LIN {X 0,Y 469.68,Z 331.264,A -85,B 0,C 180,E1 -7635.818,E2 -7635.818} C_VEL
LIN {X 0,Y 469.232,Z 342.492,A -85,B 0,C 180,E1 -7636.5,E2 -7636.5} C_VEL
LIN {X 0,Y 468.814,Z 353.33,A -85,B 0,C 180,E1 -7637.334,E2 -7637.334} C_VEL
LIN {X 0,Y 468.372,Z 363.607,A -85,B 0,C 180,E1 -7638.314,E2 -7638.314} C_VEL
LIN {X 0,Y 467.885,Z 372.795,A -85,B 0,C 180,E1 -7639.398,E2 -7639.398} C_VEL
LIN {X 0,Y 467.445,Z 381.696,A -85,B 0,C 180,E1 -7640.7,E2 -7640.7} C_VEL
LIN {X 0,Y 467.091,Z 388.855,A -85,B 0,C 180,E1 -7642.001,E2 -7642.001} C_VEL
LIN {X 0,Y 466.869,Z 395.228,A -85,B 0,C 180,E1 -7643.48,E2 -7643.48} C_VEL
LIN {X 0,Y 466.783,Z 399.68,A -85,B 0,C 180,E1 -7644.818,E2 -7644.818} C_VEL
LIN {X 0,Y 466.662,Z 401.961,A -85,B 0,C 180,E1 -7645.683,E2 -7645.683} C_VEL
LIN {X 0,Y 466.695,Z 403.809,A -85,B 0,C 180,E1 -7646.548,E2 -7646.548} C_VEL
LIN {X 0,Y 466.646,Z 405.194,A -85,B 0,C 180,E1 -7647.412,E2 -7647.412} C_VEL
LIN {X 0,Y 466.589,Z 406.786,A -85,B 0,C 180,E1 -7649.138,E2 -7649.138} C_VEL
LIN {X 0,Y 466.57,Z 407,A -85,B 0,C 180,E1 -7650.001,E2 -7650.001} C_VEL
LIN {X 0,Y 466.589,Z 406.785,A -85,B 0,C 180,E1 -7650.864,E2 -7650.864} C_VEL
LIN {X 0,Y 466.647,Z 405.194,A -85,B 0,C 180,E1 -7652.591,E2 -7652.591} C_VEL
LIN {X 0,Y 466.695,Z 403.808,A -85,B 0,C 180,E1 -7653.455,E2 -7653.455} C_VEL
LIN {X 0,Y 466.703,Z 400.892,A -85,B 0,C 180,E1 -7654.752,E2 -7654.752} C_VEL
LIN {X 0,Y 466.841,Z 396.944,A -85,B 0,C 180,E1 -7656.05,E2 -7656.05} C_VEL
LIN {X 0,Y 466.999,Z 390.87,A -85,B 0,C 180,E1 -7657.568,E2 -7657.568} C_VEL
LIN {X 0,Y 467.351,Z 384.228,A -85,B 0,C 180,E1 -7658.868,E2 -7658.868} C_VEL
LIN {X 0,Y 467.741,Z 375.984,A -85,B 0,C 180,E1 -7660.17,E2 -7660.17} C_VEL
LIN {X 0,Y 468.139,Z 367.508,A -85,B 0,C 180,E1 -7661.256,E2 -7661.256} C_VEL
LIN {X 0,Y 468.647,Z 357.179,A -85,B 0,C 180,E1 -7662.321,E2 -7662.321} C_VEL
LIN {X 0,Y 469.095,Z 345.552,A -85,B 0,C 180,E1 -7663.286,E2 -7663.286} C_VEL
LIN {X 0,Y 469.628,Z 333.213,A -85,B 0,C 180,E1 -7664.076,E2 -7664.076} C_VEL
LIN {X 0,Y 470.095,Z 320.836,A -85,B 0,C 180,E1 -7664.669,E2 -7664.669} C_VEL
LIN {X 0,Y 469.974,Z 315.841,A -85,B 0,C 180,E1 -7664.867,E2 -7664.867} C_VEL
LIN {X 0,Y 467.863,Z 303.105,A -85,B 0,C 180,E1 -7665.308,E2 -7665.308} C_VEL
LIN {X 0,Y 467.231,Z 299.138,A -85,B 0,C 180,E1 -7665.431,E2 -7665.431} C_VEL
LIN {X 0,Y 467.48,Z 289.181,A -85,B 0,C 180,E1 -7668.714,E2 -7668.714} C_VEL
LIN {X 0,Y 467.722,Z 280.399,A -85,B 0,C 180,E1 -7671.635,E2 -7671.635} C_VEL
LIN {X 0,Y 468.018,Z 270.988,A -85,B 0,C 180,E1 -7674.865,E2 -7674.865} C_VEL
LIN {X 0,Y 468.41,Z 262.951,A -85,B 0,C 180,E1 -7677.719,E2 -7677.719} C_VEL
LIN {X 0,Y 468.808,Z 253.122,A -85,B 0,C 180,E1 -7681.295,E2 -7681.295} C_VEL
LIN {X 0,Y 469.227,Z 244.558,A -85,B 0,C 180,E1 -7684.535,E2 -7684.535} C_VEL
LIN {X 0,Y 469.326,Z 240.72,A -85,B 0,C 180,E1 -7686.037,E2 -7686.037} C_VEL
LIN {X 0,Y 468.333,Z 234.391,A -85,B 0,C 180,E1 -7688.709,E2 -7688.709} C_VEL
LIN {X 0,Y 467.562,Z 230.247,A -85,B 0,C 180,E1 -7690.621,E2 -7690.621} C_VEL
LIN {X 0,Y 467.563,Z 230.248,A -85,B 0,C 180,E1 -7693.745,E2 -7693.745} C_VEL
LIN {X 0,Y 467.563,Z 230.245,A -85,B 0,C 180,E1 -7696.256,E2 -7696.256} C_VEL
LIN {X 0,Y 467.585,Z 230.241,A -85,B 0,C 180,E1 -7698.724,E2 -7698.724} C_VEL
LIN {X 0,Y 467.567,Z 230.241,A -85,B 0,C 180,E1 -7701.956,E2 -7701.956} C_VEL
LIN {X 0,Y 467.56,Z 230.241,A -85,B 0,C 180,E1 -7705.167,E2 -7705.167} C_VEL
LIN {X 0,Y 467.579,Z 230.244,A -85,B 0,C 180,E1 -7708.26,E2 -7708.26} C_VEL
LIN {X 0,Y 467.562,Z 230.243,A -85,B 0,C 180,E1 -7711.249,E2 -7711.249} C_VEL
LIN {X 0,Y 467.592,Z 230.24,A -85,B 0,C 180,E1 -7714.159,E2 -7714.159} C_VEL
LIN {X 0,Y 467.583,Z 230.241,A -85,B 0,C 180,E1 -7716.996,E2 -7716.996} C_VEL
LIN {X 0,Y 467.628,Z 230.235,A -85,B 0,C 180,E1 -7719.777,E2 -7719.777} C_VEL
LIN {X 0,Y 467.574,Z 230.243,A -85,B 0,C 180,E1 -7722.505,E2 -7722.505} C_VEL
LIN {X 0,Y 467.594,Z 230.237,A -85,B 0,C 180,E1 -7725.196,E2 -7725.196} C_VEL
LIN {X 0,Y 467.654,Z 230.235,A -85,B 0,C 180,E1 -7727.855,E2 -7727.855} C_VEL
LIN {X 0,Y 467.667,Z 230.232,A -85,B 0,C 180,E1 -7731.357,E2 -7731.357} C_VEL
LIN {X 0,Y 467.74,Z 230.221,A -85,B 0,C 180,E1 -7733.963,E2 -7733.963} C_VEL
LIN {X 0,Y 467.865,Z 230.206,A -85,B 0,C 180,E1 -7737.417,E2 -7737.417} C_VEL
LIN {X 0,Y 467.887,Z 230.205,A -85,B 0,C 180,E1 -7740,E2 -7740} C_VEL
LIN {X 0,Y 467.855,Z 230.206,A -85,B 0,C 180,E1 -7742.583,E2 -7742.583} C_VEL
LIN {X 0,Y 467.699,Z 230.224,A -85,B 0,C 180,E1 -7746.038,E2 -7746.038} C_VEL
LIN {X 0,Y 467.663,Z 230.23,A -85,B 0,C 180,E1 -7748.643,E2 -7748.643} C_VEL
LIN {X 0,Y 467.663,Z 230.23,A -85,B 0,C 180,E1 -7752.145,E2 -7752.145} C_VEL
LIN {X 0,Y 467.647,Z 230.234,A -85,B 0,C 180,E1 -7755.695,E2 -7755.695} C_VEL
LIN {X 0,Y 467.63,Z 230.237,A -85,B 0,C 180,E1 -7759.308,E2 -7759.308} C_VEL
LIN {X 0,Y 467.538,Z 230.246,A -85,B 0,C 180,E1 -7762.074,E2 -7762.074} C_VEL
LIN {X 0,Y 467.556,Z 230.248,A -85,B 0,C 180,E1 -7764.89,E2 -7764.89} C_VEL
LIN {X 0,Y 467.549,Z 230.242,A -85,B 0,C 180,E1 -7767.774,E2 -7767.774} C_VEL
LIN {X 0,Y 467.573,Z 230.241,A -85,B 0,C 180,E1 -7771.044,E2 -7771.044} C_VEL
LIN {X 0,Y 467.584,Z 230.243,A -85,B 0,C 180,E1 -7774.24,E2 -7774.24} C_VEL
LIN {X 0,Y 467.55,Z 230.246,A -85,B 0,C 180,E1 -7777.185,E2 -7777.185} C_VEL
LIN {X 0,Y 467.577,Z 230.242,A -85,B 0,C 180,E1 -7780.265,E2 -7780.265} C_VEL
LIN {X 0,Y 467.555,Z 230.243,A -85,B 0,C 180,E1 -7783.745,E2 -7783.745} C_VEL
LIN {X 0,Y 467.547,Z 230.249,A -85,B 0,C 180,E1 -7786.253,E2 -7786.253} C_VEL
LIN {X 0,Y 467.546,Z 230.247,A -85,B 0,C 180,E1 -7789.731,E2 -7789.731} C_VEL
LIN {X 0,Y 467.549,Z 230.245,A -85,B 0,C 180,E1 -7792.814,E2 -7792.814} C_VEL
LIN {X 0,Y 467.584,Z 230.241,A -85,B 0,C 180,E1 -7795.759,E2 -7795.759} C_VEL
LIN {X 0,Y 467.491,Z 230.254,A -85,B 0,C 180,E1 -7798.252,E2 -7798.252} C_VEL
LIN {X 0,Y 467.193,Z 230.292,A -85,B 0,C 180,E1 -7801.223,E2 -7801.223} C_VEL
LIN {X 0,Y 467.078,Z 230.558,A -85,B 0,C 180,E1 -7802.195,E2 -7802.195} C_VEL
LIN {X 0,Y 467.063,Z 233.522,A -85,B 0,C 180,E1 -7805.081,E2 -7805.081} C_VEL
LIN {X 0,Y 466.962,Z 236.466,A -85,B 0,C 180,E1 -7807.896,E2 -7807.896} C_VEL
LIN {X 0,Y 466.922,Z 239.387,A -85,B 0,C 180,E1 -7810.661,E2 -7810.661} C_VEL
LIN {X 0,Y 466.929,Z 242.317,A -85,B 0,C 180,E1 -7813.381,E2 -7813.381} C_VEL
LIN {X 0,Y 466.931,Z 244.335,A -85,B 0,C 180,E1 -7815.212,E2 -7815.212} C_VEL
LIN {X 0,Y 466.213,Z 244.933,A -85,B 0,C 180,E1 -7815.687,E2 -7815.687} C_VEL
LIN {X 0,Y 460.495,Z 247.155,A -85,B 0,C 180,E1 -7817.175,E2 -7817.175} C_VEL
LIN {X 0,Y 459.851,Z 247.772,A -85,B 0,C 180,E1 -7817.66,E2 -7817.66} C_VEL
LIN {X 0,Y 459.867,Z 248.764,A -85,B 0,C 180,E1 -7818.514,E2 -7818.514} C_VEL
LIN {X 0,Y 463.083,Z 262.929,A -85,B 0,C 180,E1 -7819.063,E2 -7819.063} C_VEL
LIN {X 0,Y 463.454,Z 265.604,A -85,B 0,C 180,E1 -7819.183,E2 -7819.183} C_VEL
LIN {X 0,Y 463.136,Z 277.009,A -85,B 0,C 180,E1 -7819.728,E2 -7819.728} C_VEL
LIN {X 0,Y 462.661,Z 289.11,A -85,B 0,C 180,E1 -7820.49,E2 -7820.49} C_VEL
LIN {X 0,Y 462.117,Z 299.456,A -85,B 0,C 180,E1 -7821.319,E2 -7821.319} C_VEL
LIN {X 0,Y 461.72,Z 309.658,A -85,B 0,C 180,E1 -7822.345,E2 -7822.345} C_VEL
LIN {X 0,Y 461.296,Z 318.522,A -85,B 0,C 180,E1 -7823.438,E2 -7823.438} C_VEL
LIN {X 0,Y 460.755,Z 327.192,A -85,B 0,C 180,E1 -7824.748,E2 -7824.748} C_VEL
LIN {X 0,Y 460.329,Z 334.13,A -85,B 0,C 180,E1 -7826.059,E2 -7826.059} C_VEL
LIN {X 0,Y 459.91,Z 339.682,A -85,B 0,C 180,E1 -7827.371,E2 -7827.371} C_VEL
LIN {X 0,Y 459.875,Z 344.034,A -85,B 0,C 180,E1 -7828.685,E2 -7828.685} C_VEL
LIN {X 0,Y 459.615,Z 347.358,A -85,B 0,C 180,E1 -7829.999,E2 -7829.999} C_VEL
LIN {X 0,Y 459.645,Z 350.251,A -85,B 0,C 180,E1 -7831.751,E2 -7831.751} C_VEL
LIN {X 0,Y 459.716,Z 351.112,A -85,B 0,C 180,E1 -7832.627,E2 -7832.627} C_VEL
LIN {X 0,Y 459.725,Z 351.554,A -85,B 0,C 180,E1 -7833.504,E2 -7833.504} C_VEL
LIN {X 0,Y 459.654,Z 351.285,A -85,B 0,C 180,E1 -7835.262,E2 -7835.262} C_VEL
LIN {X 0,Y 459.716,Z 350.234,A -85,B 0,C 180,E1 -7836.431,E2 -7836.431} C_VEL
LIN {X 0,Y 459.78,Z 347.889,A -85,B 0,C 180,E1 -7837.906,E2 -7837.906} C_VEL
LIN {X 0,Y 459.922,Z 344.761,A -85,B 0,C 180,E1 -7839.232,E2 -7839.232} C_VEL
LIN {X 0,Y 460.064,Z 340.568,A -85,B 0,C 180,E1 -7840.561,E2 -7840.561} C_VEL
LIN {X 0,Y 460.352,Z 335.18,A -85,B 0,C 180,E1 -7841.892,E2 -7841.892} C_VEL
LIN {X 0,Y 460.736,Z 328.418,A -85,B 0,C 180,E1 -7843.225,E2 -7843.225} C_VEL
LIN {X 0,Y 461.241,Z 319.957,A -85,B 0,C 180,E1 -7844.56,E2 -7844.56} C_VEL
LIN {X 0,Y 461.723,Z 311.216,A -85,B 0,C 180,E1 -7845.673,E2 -7845.673} C_VEL
LIN {X 0,Y 462.278,Z 300.416,A -85,B 0,C 180,E1 -7846.788,E2 -7846.788} C_VEL
LIN {X 0,Y 462.797,Z 289.54,A -85,B 0,C 180,E1 -7847.68,E2 -7847.68} C_VEL
LIN {X 0,Y 463.287,Z 277.283,A -85,B 0,C 180,E1 -7848.46,E2 -7848.46} C_VEL
LIN {X 0,Y 463.698,Z 264.849,A -85,B 0,C 180,E1 -7849.053,E2 -7849.053} C_VEL
LIN {X 0,Y 460.758,Z 252.609,A -85,B 0,C 180,E1 -7849.58,E2 -7849.58} C_VEL
LIN {X 0,Y 459.799,Z 248.855,A -85,B 0,C 180,E1 -7849.721,E2 -7849.721} C_VEL
LIN {X 0,Y 459.847,Z 244.678,A -85,B 0,C 180,E1 -7853.508,E2 -7853.508} C_VEL
LIN {X 0,Y 459.902,Z 241.674,A -85,B 0,C 180,E1 -7856.304,E2 -7856.304} C_VEL
LIN {X 0,Y 459.979,Z 238.452,A -85,B 0,C 180,E1 -7859.436,E2 -7859.436} C_VEL
LIN {X 0,Y 460.055,Z 235.013,A -85,B 0,C 180,E1 -7862.838,E2 -7862.838} C_VEL
LIN {X 0,Y 460.14,Z 231.931,A -85,B 0,C 180,E1 -7865.952,E2 -7865.952} C_VEL
LIN {X 0,Y 460.156,Z 231.333,A -85,B 0,C 180,E1 -7866.557,E2 -7866.557} C_VEL
LIN {X 0,Y 460.4,Z 231.138,A -85,B 0,C 180,E1 -7868.875,E2 -7868.875} C_VEL
LIN {X 0,Y 460.522,Z 231.12,A -85,B 0,C 180,E1 -7871.6,E2 -7871.6} C_VEL
LIN {X 0,Y 460.51,Z 231.124,A -85,B 0,C 180,E1 -7874.587,E2 -7874.587} C_VEL
LIN {X 0,Y 460.496,Z 231.126,A -85,B 0,C 180,E1 -7877.815,E2 -7877.815} C_VEL
LIN {X 0,Y 460.531,Z 231.121,A -85,B 0,C 180,E1 -7881.102,E2 -7881.102} C_VEL
LIN {X 0,Y 460.492,Z 231.124,A -85,B 0,C 180,E1 -7883.984,E2 -7883.984} C_VEL
LIN {X 0,Y 460.519,Z 231.12,A -85,B 0,C 180,E1 -7887.069,E2 -7887.069} C_VEL
LIN {X 0,Y 460.5,Z 231.121,A -85,B 0,C 180,E1 -7889.759,E2 -7889.759} C_VEL
LIN {X 0,Y 460.574,Z 231.114,A -85,B 0,C 180,E1 -7892.756,E2 -7892.756} C_VEL
LIN {X 0,Y 460.533,Z 231.122,A -85,B 0,C 180,E1 -7895.667,E2 -7895.667} C_VEL
LIN {X 0,Y 460.511,Z 231.121,A -85,B 0,C 180,E1 -7898.577,E2 -7898.577} C_VEL
LIN {X 0,Y 460.579,Z 231.111,A -85,B 0,C 180,E1 -7901.31,E2 -7901.31} C_VEL
LIN {X 0,Y 460.593,Z 231.114,A -85,B 0,C 180,E1 -7904.058,E2 -7904.058} C_VEL
LIN {X 0,Y 460.597,Z 231.111,A -85,B 0,C 180,E1 -7907.665,E2 -7907.665} C_VEL
LIN {X 0,Y 460.615,Z 231.107,A -85,B 0,C 180,E1 -7911.223,E2 -7911.223} C_VEL
LIN {X 0,Y 460.709,Z 231.1,A -85,B 0,C 180,E1 -7913.87,E2 -7913.87} C_VEL
LIN {X 0,Y 460.814,Z 231.085,A -85,B 0,C 180,E1 -7917.377,E2 -7917.377} C_VEL
LIN {X 0,Y 460.837,Z 231.081,A -85,B 0,C 180,E1 -7920,E2 -7920} C_VEL
LIN {X 0,Y 460.814,Z 231.083,A -85,B 0,C 180,E1 -7922.622,E2 -7922.622} C_VEL
LIN {X 0,Y 460.706,Z 231.096,A -85,B 0,C 180,E1 -7926.13,E2 -7926.13} C_VEL
LIN {X 0,Y 460.616,Z 231.111,A -85,B 0,C 180,E1 -7928.776,E2 -7928.776} C_VEL
LIN {X 0,Y 460.601,Z 231.109,A -85,B 0,C 180,E1 -7932.445,E2 -7932.445} C_VEL
LIN {X 0,Y 460.588,Z 231.109,A -85,B 0,C 180,E1 -7935.998,E2 -7935.998} C_VEL
LIN {X 0,Y 460.559,Z 231.115,A -85,B 0,C 180,E1 -7938.902,E2 -7938.902} C_VEL
LIN {X 0,Y 460.504,Z 231.123,A -85,B 0,C 180,E1 -7941.486,E2 -7941.486} C_VEL
LIN {X 0,Y 460.529,Z 231.118,A -85,B 0,C 180,E1 -7944.333,E2 -7944.333} C_VEL
LIN {X 0,Y 460.574,Z 231.114,A -85,B 0,C 180,E1 -7947.244,E2 -7947.244} C_VEL
LIN {X 0,Y 460.517,Z 231.124,A -85,B 0,C 180,E1 -7950.24,E2 -7950.24} C_VEL
LIN {X 0,Y 460.519,Z 231.124,A -85,B 0,C 180,E1 -7953.326,E2 -7953.326} C_VEL
LIN {X 0,Y 460.467,Z 231.13,A -85,B 0,C 180,E1 -7956.53,E2 -7956.53} C_VEL
LIN {X 0,Y 460.524,Z 231.121,A -85,B 0,C 180,E1 -7959.863,E2 -7959.863} C_VEL
LIN {X 0,Y 460.484,Z 231.125,A -85,B 0,C 180,E1 -7962.899,E2 -7962.899} C_VEL
LIN {X 0,Y 460.504,Z 231.124,A -85,B 0,C 180,E1 -7965.832,E2 -7965.832} C_VEL
LIN {X 0,Y 460.572,Z 231.215,A -85,B 0,C 180,E1 -7968.875,E2 -7968.875} C_VEL
LIN {X 0,Y 461.492,Z 236.488,A -85,B 0,C 180,E1 -7971.365,E2 -7971.365} C_VEL
LIN {X 0,Y 462.298,Z 241.71,A -85,B 0,C 180,E1 -7973.68,E2 -7973.68} C_VEL
LIN {X 0,Y 462.271,Z 245.337,A -85,B 0,C 180,E1 -7975.183,E2 -7975.183} C_VEL
LIN {X 0,Y 461.928,Z 252.022,A -85,B 0,C 180,E1 -7977.827,E2 -7977.827} C_VEL
LIN {X 0,Y 461.451,Z 259.973,A -85,B 0,C 180,E1 -7980.834,E2 -7980.834} C_VEL
LIN {X 0,Y 461.172,Z 268.023,A -85,B 0,C 180,E1 -7983.774,E2 -7983.774} C_VEL
LIN {X 0,Y 460.776,Z 277.442,A -85,B 0,C 180,E1 -7987.113,E2 -7987.113} C_VEL
LIN {X 0,Y 460.491,Z 287,A -85,B 0,C 180,E1 -7990.383,E2 -7990.383} C_VEL
LIN {X 0,Y 460.175,Z 296.503,A -85,B 0,C 180,E1 -7993.59,E2 -7993.59} C_VEL
LIN {X 0,Y 460.16,Z 298.734,A -85,B 0,C 180,E1 -7994.341,E2 -7994.341} C_VEL
LIN {X 0,Y 462.493,Z 312.669,A -85,B 0,C 180,E1 -7994.788,E2 -7994.788} C_VEL
LIN {X 0,Y 463.231,Z 319.164,A -85,B 0,C 180,E1 -7995.055,E2 -7995.055} C_VEL
LIN {X 0,Y 462.811,Z 330.833,A -85,B 0,C 180,E1 -7995.603,E2 -7995.603} C_VEL
LIN {X 0,Y 462.258,Z 343.171,A -85,B 0,C 180,E1 -7996.371,E2 -7996.371} C_VEL
LIN {X 0,Y 461.804,Z 353.442,A -85,B 0,C 180,E1 -7997.185,E2 -7997.185} C_VEL
LIN {X 0,Y 461.363,Z 363.172,A -85,B 0,C 180,E1 -7998.134,E2 -7998.134} C_VEL
LIN {X 0,Y 460.872,Z 372.39,A -85,B 0,C 180,E1 -7999.235,E2 -7999.235} C_VEL
LIN {X 0,Y 460.415,Z 381.379,A -85,B 0,C 180,E1 -8000.557,E2 -8000.557} C_VEL
LIN {X 0,Y 460.053,Z 388.617,A -85,B 0,C 180,E1 -8001.878,E2 -8001.878} C_VEL
LIN {X 0,Y 459.846,Z 393.507,A -85,B 0,C 180,E1 -8002.978,E2 -8002.978} C_VEL
LIN {X 0,Y 459.755,Z 398.267,A -85,B 0,C 180,E1 -8004.299,E2 -8004.299} C_VEL
LIN {X 0,Y 459.579,Z 401.898,A -85,B 0,C 180,E1 -8005.616,E2 -8005.616} C_VEL
LIN {X 0,Y 459.591,Z 403.776,A -85,B 0,C 180,E1 -8006.494,E2 -8006.494} C_VEL
LIN {X 0,Y 459.57,Z 405.177,A -85,B 0,C 180,E1 -8007.372,E2 -8007.372} C_VEL
LIN {X 0,Y 459.494,Z 406.779,A -85,B 0,C 180,E1 -8009.125,E2 -8009.125} C_VEL
LIN {X 0,Y 459.474,Z 406.994,A -85,B 0,C 180,E1 -8010.001,E2 -8010.001} C_VEL
LIN {X 0,Y 459.494,Z 406.778,A -85,B 0,C 180,E1 -8010.878,E2 -8010.878} C_VEL
LIN {X 0,Y 459.571,Z 405.177,A -85,B 0,C 180,E1 -8012.631,E2 -8012.631} C_VEL
LIN {X 0,Y 459.591,Z 403.774,A -85,B 0,C 180,E1 -8013.508,E2 -8013.508} C_VEL
LIN {X 0,Y 459.635,Z 400.815,A -85,B 0,C 180,E1 -8014.825,E2 -8014.825} C_VEL
LIN {X 0,Y 459.759,Z 396.813,A -85,B 0,C 180,E1 -8016.144,E2 -8016.144} C_VEL
LIN {X 0,Y 459.93,Z 390.656,A -85,B 0,C 180,E1 -8017.685,E2 -8017.685} C_VEL
LIN {X 0,Y 460.288,Z 383.942,A -85,B 0,C 180,E1 -8019.005,E2 -8019.005} C_VEL
LIN {X 0,Y 460.705,Z 375.613,A -85,B 0,C 180,E1 -8020.327,E2 -8020.327} C_VEL
LIN {X 0,Y 461.142,Z 367.081,A -85,B 0,C 180,E1 -8021.429,E2 -8021.429} C_VEL
LIN {X 0,Y 461.652,Z 356.921,A -85,B 0,C 180,E1 -8022.495,E2 -8022.495} C_VEL
LIN {X 0,Y 462.116,Z 346.127,A -85,B 0,C 180,E1 -8023.412,E2 -8023.412} C_VEL
LIN {X 0,Y 462.639,Z 334.717,A -85,B 0,C 180,E1 -8024.18,E2 -8024.18} C_VEL
LIN {X 0,Y 463.115,Z 323.017,A -85,B 0,C 180,E1 -8024.783,E2 -8024.783} C_VEL
LIN {X 0,Y 463.058,Z 316.605,A -85,B 0,C 180,E1 -8025.05,E2 -8025.05} C_VEL
LIN {X 0,Y 460.792,Z 302.902,A -85,B 0,C 180,E1 -8025.543,E2 -8025.543} C_VEL
LIN {X 0,Y 460.172,Z 298.742,A -85,B 0,C 180,E1 -8025.663,E2 -8025.663} C_VEL
LIN {X 0,Y 460.449,Z 288.329,A -85,B 0,C 180,E1 -8029.179,E2 -8029.179} C_VEL
LIN {X 0,Y 460.73,Z 278.815,A -85,B 0,C 180,E1 -8032.419,E2 -8032.419} C_VEL
LIN {X 0,Y 461.118,Z 268.862,A -85,B 0,C 180,E1 -8035.942,E2 -8035.942} C_VEL
LIN {X 0,Y 461.424,Z 261.324,A -85,B 0,C 180,E1 -8038.672,E2 -8038.672} C_VEL
LIN {X 0,Y 461.828,Z 253.601,A -85,B 0,C 180,E1 -8041.549,E2 -8041.549} C_VEL
LIN {X 0,Y 462.273,Z 245.106,A -85,B 0,C 180,E1 -8044.818,E2 -8044.818} C_VEL
LIN {X 0,Y 462.25,Z 241.264,A -85,B 0,C 180,E1 -8046.368,E2 -8046.368} C_VEL
LIN {X 0,Y 461.27,Z 235.139,A -85,B 0,C 180,E1 -8049.009,E2 -8049.009} C_VEL
LIN {X 0,Y 460.541,Z 231.121,A -85,B 0,C 180,E1 -8050.913,E2 -8050.913} C_VEL
LIN {X 0,Y 460.518,Z 231.126,A -85,B 0,C 180,E1 -8054.17,E2 -8054.17} C_VEL
LIN {X 0,Y 460.52,Z 231.122,A -85,B 0,C 180,E1 -8057.1,E2 -8057.1} C_VEL
LIN {X 0,Y 460.532,Z 231.118,A -85,B 0,C 180,E1 -8060.138,E2 -8060.138} C_VEL
LIN {X 0,Y 460.477,Z 231.124,A -85,B 0,C 180,E1 -8063.471,E2 -8063.471} C_VEL
LIN {X 0,Y 460.522,Z 231.122,A -85,B 0,C 180,E1 -8066.674,E2 -8066.674} C_VEL
LIN {X 0,Y 460.511,Z 231.121,A -85,B 0,C 180,E1 -8069.76,E2 -8069.76} C_VEL
LIN {X 0,Y 460.542,Z 231.118,A -85,B 0,C 180,E1 -8072.754,E2 -8072.754} C_VEL
LIN {X 0,Y 460.536,Z 231.12,A -85,B 0,C 180,E1 -8075.667,E2 -8075.667} C_VEL
LIN {X 0,Y 460.529,Z 231.122,A -85,B 0,C 180,E1 -8078.579,E2 -8078.579} C_VEL
LIN {X 0,Y 460.59,Z 231.111,A -85,B 0,C 180,E1 -8081.311,E2 -8081.311} C_VEL
LIN {X 0,Y 460.574,Z 231.117,A -85,B 0,C 180,E1 -8084.058,E2 -8084.058} C_VEL
LIN {X 0,Y 460.609,Z 231.111,A -85,B 0,C 180,E1 -8087.666,E2 -8087.666} C_VEL
LIN {X 0,Y 460.614,Z 231.109,A -85,B 0,C 180,E1 -8091.224,E2 -8091.224} C_VEL
LIN {X 0,Y 460.706,Z 231.097,A -85,B 0,C 180,E1 -8093.87,E2 -8093.87} C_VEL
LIN {X 0,Y 460.806,Z 231.085,A -85,B 0,C 180,E1 -8097.378,E2 -8097.378} C_VEL
LIN {X 0,Y 460.857,Z 231.08,A -85,B 0,C 180,E1 -8100,E2 -8100} C_VEL
LIN {X 0,Y 460.795,Z 231.085,A -85,B 0,C 180,E1 -8102.623,E2 -8102.623} C_VEL
LIN {X 0,Y 460.666,Z 231.099,A -85,B 0,C 180,E1 -8106.131,E2 -8106.131} C_VEL
LIN {X 0,Y 460.613,Z 231.109,A -85,B 0,C 180,E1 -8108.777,E2 -8108.777} C_VEL
LIN {X 0,Y 460.617,Z 231.108,A -85,B 0,C 180,E1 -8112.334,E2 -8112.334} C_VEL
LIN {X 0,Y 460.609,Z 231.11,A -85,B 0,C 180,E1 -8115.997,E2 -8115.997} C_VEL
LIN {X 0,Y 460.576,Z 231.114,A -85,B 0,C 180,E1 -8119.615,E2 -8119.615} C_VEL
LIN {X 0,Y 460.514,Z 231.12,A -85,B 0,C 180,E1 -8122.429,E2 -8122.429} C_VEL
LIN {X 0,Y 460.528,Z 231.117,A -85,B 0,C 180,E1 -8125.789,E2 -8125.789} C_VEL
LIN {X 0,Y 460.527,Z 231.118,A -85,B 0,C 180,E1 -8129.232,E2 -8129.232} C_VEL
LIN {X 0,Y 460.537,Z 231.122,A -85,B 0,C 180,E1 -8132.284,E2 -8132.284} C_VEL
LIN {X 0,Y 460.514,Z 231.121,A -85,B 0,C 180,E1 -8135.446,E2 -8135.446} C_VEL
LIN {X 0,Y 460.538,Z 231.12,A -85,B 0,C 180,E1 -8138.895,E2 -8138.895} C_VEL
LIN {X 0,Y 460.511,Z 231.122,A -85,B 0,C 180,E1 -8142.183,E2 -8142.183} C_VEL
LIN {X 0,Y 460.516,Z 231.119,A -85,B 0,C 180,E1 -8145.41,E2 -8145.41} C_VEL
LIN {X 0,Y 460.51,Z 231.119,A -85,B 0,C 180,E1 -8148.985,E2 -8148.985} C_VEL
LIN {X 0,Y 460.505,Z 231.122,A -85,B 0,C 180,E1 -8152.376,E2 -8152.376} C_VEL
LIN {X 0,Y 460.543,Z 231.119,A -85,B 0,C 180,E1 -8155.622,E2 -8155.622} C_VEL
LIN {X 0,Y 460.482,Z 231.125,A -85,B 0,C 180,E1 -8157.71,E2 -8157.71} C_VEL
LIN {X 0,Y 460.236,Z 231.157,A -85,B 0,C 180,E1 -8160.747,E2 -8160.747} C_VEL
LIN {X 0,Y 460.025,Z 231.504,A -85,B 0,C 180,E1 -8162.387,E2 -8162.387} C_VEL
LIN {X 0,Y 459.986,Z 234.841,A -85,B 0,C 180,E1 -8165.635,E2 -8165.635} C_VEL
LIN {X 0,Y 459.913,Z 238.097,A -85,B 0,C 180,E1 -8168.774,E2 -8168.774} C_VEL
LIN {X 0,Y 459.869,Z 241.714,A -85,B 0,C 180,E1 -8172.201,E2 -8172.201} C_VEL
LIN {X 0,Y 459.846,Z 244.981,A -85,B 0,C 180,E1 -8175.192,E2 -8175.192} C_VEL
LIN {X 0,Y 459.851,Z 247.772,A -85,B 0,C 180,E1 -8177.66,E2 -8177.66} C_VEL
LIN {X 0,Y 459.786,Z 248.948,A -85,B 0,C 180,E1 -8178.007,E2 -8178.007} C_VEL
LIN {X 0,Y 459.494,Z 251.95,A -85,B 0,C 180,E1 -8178.361,E2 -8178.361} C_VEL
LIN {X 0,Y 458.898,Z 256.941,A -85,B 0,C 180,E1 -8178.663,E2 -8178.663} C_VEL
LIN {X 0,Y 456.606,Z 272.462,A -85,B 0,C 180,E1 -8179.264,E2 -8179.264} C_VEL
LIN {X 0,Y 456.325,Z 275.978,A -85,B 0,C 180,E1 -8179.443,E2 -8179.443} C_VEL
LIN {X 0,Y 455.886,Z 287.069,A -85,B 0,C 180,E1 -8180.123,E2 -8180.123} C_VEL
LIN {X 0,Y 455.289,Z 298.369,A -85,B 0,C 180,E1 -8181.007,E2 -8181.007} C_VEL
LIN {X 0,Y 454.842,Z 308.54,A -85,B 0,C 180,E1 -8182.005,E2 -8182.005} C_VEL
LIN {X 0,Y 454.366,Z 317.688,A -85,B 0,C 180,E1 -8183.114,E2 -8183.114} C_VEL
LIN {X 0,Y 453.834,Z 326.566,A -85,B 0,C 180,E1 -8184.445,E2 -8184.445} C_VEL
LIN {X 0,Y 453.38,Z 333.724,A -85,B 0,C 180,E1 -8185.776,E2 -8185.776} C_VEL
LIN {X 0,Y 453.049,Z 338.569,A -85,B 0,C 180,E1 -8186.886,E2 -8186.886} C_VEL
LIN {X 0,Y 452.711,Z 343.283,A -85,B 0,C 180,E1 -8188.219,E2 -8188.219} C_VEL
LIN {X 0,Y 452.685,Z 346.885,A -85,B 0,C 180,E1 -8189.554,E2 -8189.554} C_VEL
LIN {X 0,Y 452.522,Z 349.507,A -85,B 0,C 180,E1 -8190.889,E2 -8190.889} C_VEL
LIN {X 0,Y 452.585,Z 350.736,A -85,B 0,C 180,E1 -8191.778,E2 -8191.778} C_VEL
LIN {X 0,Y 452.634,Z 351.575,A -85,B 0,C 180,E1 -8192.669,E2 -8192.669} C_VEL
LIN {X 0,Y 452.654,Z 351.988,A -85,B 0,C 180,E1 -8193.559,E2 -8193.559} C_VEL
LIN {X 0,Y 452.592,Z 351.685,A -85,B 0,C 180,E1 -8195.345,E2 -8195.345} C_VEL
LIN {X 0,Y 452.651,Z 350.715,A -85,B 0,C 180,E1 -8196.439,E2 -8196.439} C_VEL
LIN {X 0,Y 452.73,Z 348.221,A -85,B 0,C 180,E1 -8198.03,E2 -8198.03} C_VEL
LIN {X 0,Y 452.871,Z 345.055,A -85,B 0,C 180,E1 -8199.377,E2 -8199.377} C_VEL
LIN {X 0,Y 453.055,Z 340.822,A -85,B 0,C 180,E1 -8200.727,E2 -8200.727} C_VEL
LIN {X 0,Y 453.339,Z 335.491,A -85,B 0,C 180,E1 -8202.057,E2 -8202.057} C_VEL
LIN {X 0,Y 453.778,Z 328.583,A -85,B 0,C 180,E1 -8203.432,E2 -8203.432} C_VEL
LIN {X 0,Y 454.207,Z 321.607,A -85,B 0,C 180,E1 -8204.561,E2 -8204.561} C_VEL
LIN {X 0,Y 454.717,Z 313.172,A -85,B 0,C 180,E1 -8205.691,E2 -8205.691} C_VEL
LIN {X 0,Y 455.248,Z 304.303,A -85,B 0,C 180,E1 -8206.667,E2 -8206.667} C_VEL
LIN {X 0,Y 455.771,Z 293.726,A -85,B 0,C 180,E1 -8207.613,E2 -8207.613} C_VEL
LIN {X 0,Y 456.319,Z 282.62,A -85,B 0,C 180,E1 -8208.403,E2 -8208.403} C_VEL
LIN {X 0,Y 456.683,Z 271.039,A -85,B 0,C 180,E1 -8209.045,E2 -8209.045} C_VEL
LIN {X 0,Y 456.798,Z 265.609,A -85,B 0,C 180,E1 -8209.288,E2 -8209.288} C_VEL
LIN {X 0,Y 453.697,Z 253.03,A -85,B 0,C 180,E1 -8209.847,E2 -8209.847} C_VEL
LIN {X 0,Y 452.732,Z 249.262,A -85,B 0,C 180,E1 -8209.997,E2 -8209.997} C_VEL
LIN {X 0,Y 452.789,Z 245.098,A -85,B 0,C 180,E1 -8213.799,E2 -8213.799} C_VEL
LIN {X 0,Y 452.846,Z 241.963,A -85,B 0,C 180,E1 -8216.746,E2 -8216.746} C_VEL
LIN {X 0,Y 452.928,Z 238.884,A -85,B 0,C 180,E1 -8219.769,E2 -8219.769} C_VEL
LIN {X 0,Y 452.998,Z 235.562,A -85,B 0,C 180,E1 -8223.093,E2 -8223.093} C_VEL
LIN {X 0,Y 453.112,Z 232.468,A -85,B 0,C 180,E1 -8226.24,E2 -8226.24} C_VEL
LIN {X 0,Y 453.237,Z 232.031,A -85,B 0,C 180,E1 -8227.738,E2 -8227.738} C_VEL
LIN {X 0,Y 453.462,Z 231.999,A -85,B 0,C 180,E1 -8230.61,E2 -8230.61} C_VEL
LIN {X 0,Y 453.45,Z 232.001,A -85,B 0,C 180,E1 -8233.243,E2 -8233.243} C_VEL
LIN {X 0,Y 453.456,Z 232.003,A -85,B 0,C 180,E1 -8235.777,E2 -8235.777} C_VEL
LIN {X 0,Y 453.486,Z 232,A -85,B 0,C 180,E1 -8239.408,E2 -8239.408} C_VEL
LIN {X 0,Y 453.462,Z 232,A -85,B 0,C 180,E1 -8242.811,E2 -8242.811} C_VEL
LIN {X 0,Y 453.468,Z 232,A -85,B 0,C 180,E1 -8246.086,E2 -8246.086} C_VEL
LIN {X 0,Y 453.467,Z 232,A -85,B 0,C 180,E1 -8249.239,E2 -8249.239} C_VEL
LIN {X 0,Y 453.534,Z 231.992,A -85,B 0,C 180,E1 -8252.297,E2 -8252.297} C_VEL
LIN {X 0,Y 453.504,Z 231.994,A -85,B 0,C 180,E1 -8255.265,E2 -8255.265} C_VEL
LIN {X 0,Y 453.469,Z 231.998,A -85,B 0,C 180,E1 -8258.414,E2 -8258.414} C_VEL
LIN {X 0,Y 453.511,Z 231.994,A -85,B 0,C 180,E1 -8261.008,E2 -8261.008} C_VEL
LIN {X 0,Y 453.557,Z 231.99,A -85,B 0,C 180,E1 -8263.879,E2 -8263.879} C_VEL
LIN {X 0,Y 453.552,Z 231.99,A -85,B 0,C 180,E1 -8267.471,E2 -8267.471} C_VEL
LIN {X 0,Y 453.578,Z 231.985,A -85,B 0,C 180,E1 -8271.086,E2 -8271.086} C_VEL
LIN {X 0,Y 453.674,Z 231.975,A -85,B 0,C 180,E1 -8273.775,E2 -8273.775} C_VEL
LIN {X 0,Y 453.755,Z 231.965,A -85,B 0,C 180,E1 -8277.337,E2 -8277.337} C_VEL
LIN {X 0,Y 453.808,Z 231.956,A -85,B 0,C 180,E1 -8280,E2 -8280} C_VEL
LIN {X 0,Y 453.754,Z 231.963,A -85,B 0,C 180,E1 -8282.663,E2 -8282.663} C_VEL
LIN {X 0,Y 453.673,Z 231.972,A -85,B 0,C 180,E1 -8286.225,E2 -8286.225} C_VEL
LIN {X 0,Y 453.58,Z 231.987,A -85,B 0,C 180,E1 -8288.914,E2 -8288.914} C_VEL
LIN {X 0,Y 453.551,Z 231.987,A -85,B 0,C 180,E1 -8292.529,E2 -8292.529} C_VEL
LIN {X 0,Y 453.533,Z 231.987,A -85,B 0,C 180,E1 -8296.196,E2 -8296.196} C_VEL
LIN {X 0,Y 453.509,Z 231.992,A -85,B 0,C 180,E1 -8299.041,E2 -8299.041} C_VEL
LIN {X 0,Y 453.465,Z 232.002,A -85,B 0,C 180,E1 -8301.837,E2 -8301.837} C_VEL
LIN {X 0,Y 453.502,Z 231.994,A -85,B 0,C 180,E1 -8304.735,E2 -8304.735} C_VEL
LIN {X 0,Y 453.529,Z 231.991,A -85,B 0,C 180,E1 -8307.962,E2 -8307.962} C_VEL
LIN {X 0,Y 453.473,Z 231.997,A -85,B 0,C 180,E1 -8310.76,E2 -8310.76} C_VEL
LIN {X 0,Y 453.467,Z 232,A -85,B 0,C 180,E1 -8313.914,E2 -8313.914} C_VEL
LIN {X 0,Y 453.443,Z 232.001,A -85,B 0,C 180,E1 -8317.191,E2 -8317.191} C_VEL
LIN {X 0,Y 453.481,Z 231.997,A -85,B 0,C 180,E1 -8319.451,E2 -8319.451} C_VEL
LIN {X 0,Y 453.452,Z 232.003,A -85,B 0,C 180,E1 -8321.934,E2 -8321.934} C_VEL
LIN {X 0,Y 453.479,Z 231.999,A -85,B 0,C 180,E1 -8325.472,E2 -8325.472} C_VEL
LIN {X 0,Y 453.493,Z 232.062,A -85,B 0,C 180,E1 -8328.51,E2 -8328.51} C_VEL
LIN {X 0,Y 454.518,Z 237.717,A -85,B 0,C 180,E1 -8331.241,E2 -8331.241} C_VEL
LIN {X 0,Y 455.288,Z 242.455,A -85,B 0,C 180,E1 -8333.388,E2 -8333.388} C_VEL
LIN {X 0,Y 455.283,Z 246.662,A -85,B 0,C 180,E1 -8335.171,E2 -8335.171} C_VEL
LIN {X 0,Y 454.843,Z 254.489,A -85,B 0,C 180,E1 -8338.31,E2 -8338.31} C_VEL
LIN {X 0,Y 454.373,Z 263.731,A -85,B 0,C 180,E1 -8341.842,E2 -8341.842} C_VEL
LIN {X 0,Y 453.972,Z 271.774,A -85,B 0,C 180,E1 -8344.805,E2 -8344.805} C_VEL
LIN {X 0,Y 453.597,Z 281.762,A -85,B 0,C 180,E1 -8348.379,E2 -8348.379} C_VEL
LIN {X 0,Y 453.288,Z 290.664,A -85,B 0,C 180,E1 -8351.476,E2 -8351.476} C_VEL
LIN {X 0,Y 453.074,Z 298.321,A -85,B 0,C 180,E1 -8354.099,E2 -8354.099} C_VEL
LIN {X 0,Y 455.175,Z 311.061,A -85,B 0,C 180,E1 -8354.501,E2 -8354.501} C_VEL
LIN {X 0,Y 456.297,Z 320.034,A -85,B 0,C 180,E1 -8354.879,E2 -8354.879} C_VEL
LIN {X 0,Y 455.813,Z 332.393,A -85,B 0,C 180,E1 -8355.491,E2 -8355.491} C_VEL
LIN {X 0,Y 455.269,Z 344.282,A -85,B 0,C 180,E1 -8356.272,E2 -8356.272} C_VEL
LIN {X 0,Y 454.744,Z 354.97,A -85,B 0,C 180,E1 -8357.167,E2 -8357.167} C_VEL
LIN {X 0,Y 454.267,Z 364.706,A -85,B 0,C 180,E1 -8358.172,E2 -8358.172} C_VEL
LIN {X 0,Y 453.734,Z 373.596,A -85,B 0,C 180,E1 -8359.289,E2 -8359.289} C_VEL
LIN {X 0,Y 453.307,Z 382.277,A -85,B 0,C 180,E1 -8360.633,E2 -8360.633} C_VEL
LIN {X 0,Y 452.923,Z 389.216,A -85,B 0,C 180,E1 -8361.974,E2 -8361.974} C_VEL
LIN {X 0,Y 452.709,Z 395.44,A -85,B 0,C 180,E1 -8363.494,E2 -8363.494} C_VEL
LIN {X 0,Y 452.566,Z 400.392,A -85,B 0,C 180,E1 -8365.102,E2 -8365.102} C_VEL
LIN {X 0,Y 452.493,Z 403.347,A -85,B 0,C 180,E1 -8366.439,E2 -8366.439} C_VEL
LIN {X 0,Y 452.495,Z 404.756,A -85,B 0,C 180,E1 -8367.331,E2 -8367.331} C_VEL
LIN {X 0,Y 452.433,Z 406.371,A -85,B 0,C 180,E1 -8369.111,E2 -8369.111} C_VEL
LIN {X 0,Y 452.41,Z 406.588,A -85,B 0,C 180,E1 -8370.001,E2 -8370.001} C_VEL
LIN {X 0,Y 452.433,Z 406.371,A -85,B 0,C 180,E1 -8370.891,E2 -8370.891} C_VEL
LIN {X 0,Y 452.496,Z 404.757,A -85,B 0,C 180,E1 -8372.672,E2 -8372.672} C_VEL
LIN {X 0,Y 452.494,Z 403.348,A -85,B 0,C 180,E1 -8373.563,E2 -8373.563} C_VEL
LIN {X 0,Y 452.567,Z 400.389,A -85,B 0,C 180,E1 -8374.901,E2 -8374.901} C_VEL
LIN {X 0,Y 452.692,Z 395.511,A -85,B 0,C 180,E1 -8376.487,E2 -8376.487} C_VEL
LIN {X 0,Y 452.927,Z 389.211,A -85,B 0,C 180,E1 -8378.029,E2 -8378.029} C_VEL
LIN {X 0,Y 453.311,Z 382.27,A -85,B 0,C 180,E1 -8379.37,E2 -8379.37} C_VEL
LIN {X 0,Y 453.736,Z 373.587,A -85,B 0,C 180,E1 -8380.713,E2 -8380.713} C_VEL
LIN {X 0,Y 454.273,Z 364.694,A -85,B 0,C 180,E1 -8381.83,E2 -8381.83} C_VEL
LIN {X 0,Y 454.782,Z 354.872,A -85,B 0,C 180,E1 -8382.842,E2 -8382.842} C_VEL
LIN {X 0,Y 455.288,Z 344.268,A -85,B 0,C 180,E1 -8383.73,E2 -8383.73} C_VEL
LIN {X 0,Y 455.81,Z 332.359,A -85,B 0,C 180,E1 -8384.512,E2 -8384.512} C_VEL
LIN {X 0,Y 456.341,Z 319.983,A -85,B 0,C 180,E1 -8385.122,E2 -8385.122} C_VEL
LIN {X 0,Y 454.873,Z 309.265,A -85,B 0,C 180,E1 -8385.565,E2 -8385.565} C_VEL
LIN {X 0,Y 453.09,Z 298.318,A -85,B 0,C 180,E1 -8385.908,E2 -8385.908} C_VEL
LIN {X 0,Y 453.412,Z 287.955,A -85,B 0,C 180,E1 -8389.468,E2 -8389.468} C_VEL
LIN {X 0,Y 453.718,Z 278.521,A -85,B 0,C 180,E1 -8392.784,E2 -8392.784} C_VEL
LIN {X 0,Y 454.126,Z 269.176,A -85,B 0,C 180,E1 -8396.155,E2 -8396.155} C_VEL
LIN {X 0,Y 454.391,Z 262.398,A -85,B 0,C 180,E1 -8398.652,E2 -8398.652} C_VEL
LIN {X 0,Y 454.834,Z 254.075,A -85,B 0,C 180,E1 -8401.805,E2 -8401.805} C_VEL
LIN {X 0,Y 455.272,Z 246.346,A -85,B 0,C 180,E1 -8404.833,E2 -8404.833} C_VEL
LIN {X 0,Y 455.222,Z 242.048,A -85,B 0,C 180,E1 -8406.601,E2 -8406.601} C_VEL
LIN {X 0,Y 454.177,Z 235.747,A -85,B 0,C 180,E1 -8409.38,E2 -8409.38} C_VEL
LIN {X 0,Y 453.499,Z 231.999,A -85,B 0,C 180,E1 -8411.197,E2 -8411.197} C_VEL
LIN {X 0,Y 453.494,Z 232,A -85,B 0,C 180,E1 -8414.53,E2 -8414.53} C_VEL
LIN {X 0,Y 453.486,Z 231.997,A -85,B 0,C 180,E1 -8418.21,E2 -8418.21} C_VEL
LIN {X 0,Y 453.496,Z 231.998,A -85,B 0,C 180,E1 -8420.795,E2 -8420.795} C_VEL
LIN {X 0,Y 453.456,Z 231.998,A -85,B 0,C 180,E1 -8423.917,E2 -8423.917} C_VEL
LIN {X 0,Y 453.479,Z 231.996,A -85,B 0,C 180,E1 -8427.151,E2 -8427.151} C_VEL
LIN {X 0,Y 453.472,Z 232.001,A -85,B 0,C 180,E1 -8430.268,E2 -8430.268} C_VEL
LIN {X 0,Y 453.479,Z 231.997,A -85,B 0,C 180,E1 -8433.292,E2 -8433.292} C_VEL
LIN {X 0,Y 453.503,Z 231.995,A -85,B 0,C 180,E1 -8436.239,E2 -8436.239} C_VEL
LIN {X 0,Y 453.489,Z 231.996,A -85,B 0,C 180,E1 -8439.118,E2 -8439.118} C_VEL
LIN {X 0,Y 453.494,Z 231.996,A -85,B 0,C 180,E1 -8441.944,E2 -8441.944} C_VEL
LIN {X 0,Y 453.524,Z 231.99,A -85,B 0,C 180,E1 -8444.726,E2 -8444.726} C_VEL
LIN {X 0,Y 453.572,Z 231.986,A -85,B 0,C 180,E1 -8447.471,E2 -8447.471} C_VEL
LIN {X 0,Y 453.579,Z 231.985,A -85,B 0,C 180,E1 -8451.086,E2 -8451.086} C_VEL
LIN {X 0,Y 453.673,Z 231.974,A -85,B 0,C 180,E1 -8453.775,E2 -8453.775} C_VEL
LIN {X 0,Y 453.75,Z 231.964,A -85,B 0,C 180,E1 -8457.337,E2 -8457.337} C_VEL
LIN {X 0,Y 453.827,Z 231.956,A -85,B 0,C 180,E1 -8460,E2 -8460} C_VEL
LIN {X 0,Y 453.739,Z 231.964,A -85,B 0,C 180,E1 -8462.663,E2 -8462.663} C_VEL
LIN {X 0,Y 453.634,Z 231.975,A -85,B 0,C 180,E1 -8466.226,E2 -8466.226} C_VEL
LIN {X 0,Y 453.579,Z 231.986,A -85,B 0,C 180,E1 -8468.914,E2 -8468.914} C_VEL
LIN {X 0,Y 453.572,Z 231.986,A -85,B 0,C 180,E1 -8472.529,E2 -8472.529} C_VEL
LIN {X 0,Y 453.553,Z 231.988,A -85,B 0,C 180,E1 -8476.196,E2 -8476.196} C_VEL
LIN {X 0,Y 453.525,Z 231.993,A -85,B 0,C 180,E1 -8479.039,E2 -8479.039} C_VEL
LIN {X 0,Y 453.483,Z 231.996,A -85,B 0,C 180,E1 -8481.836,E2 -8481.836} C_VEL
LIN {X 0,Y 453.469,Z 232.001,A -85,B 0,C 180,E1 -8484.737,E2 -8484.737} C_VEL
LIN {X 0,Y 453.467,Z 231.996,A -85,B 0,C 180,E1 -8487.942,E2 -8487.942} C_VEL
LIN {X 0,Y 453.481,Z 231.998,A -85,B 0,C 180,E1 -8490.759,E2 -8490.759} C_VEL
LIN {X 0,Y 453.476,Z 231.999,A -85,B 0,C 180,E1 -8493.913,E2 -8493.913} C_VEL
LIN {X 0,Y 453.457,Z 232.001,A -85,B 0,C 180,E1 -8497.19,E2 -8497.19} C_VEL
LIN {X 0,Y 453.501,Z 231.997,A -85,B 0,C 180,E1 -8500.609,E2 -8500.609} C_VEL
LIN {X 0,Y 453.467,Z 232.001,A -85,B 0,C 180,E1 -8504.221,E2 -8504.221} C_VEL
LIN {X 0,Y 453.425,Z 232.001,A -85,B 0,C 180,E1 -8506.999,E2 -8506.999} C_VEL
LIN {X 0,Y 453.473,Z 231.997,A -85,B 0,C 180,E1 -8509.413,E2 -8509.413} C_VEL
LIN {X 0,Y 453.456,Z 232,A -85,B 0,C 180,E1 -8512.809,E2 -8512.809} C_VEL
LIN {X 0,Y 453.47,Z 231.999,A -85,B 0,C 180,E1 -8516.085,E2 -8516.085} C_VEL
LIN {X 0,Y 453.308,Z 232.021,A -85,B 0,C 180,E1 -8519.227,E2 -8519.227} C_VEL
LIN {X 0,Y 452.968,Z 232.065,A -85,B 0,C 180,E1 -8522.176,E2 -8522.176} C_VEL
LIN {X 0,Y 452.935,Z 235.164,A -85,B 0,C 180,E1 -8525.231,E2 -8525.231} C_VEL
LIN {X 0,Y 452.841,Z 238.649,A -85,B 0,C 180,E1 -8528.622,E2 -8528.622} C_VEL
LIN {X 0,Y 452.803,Z 242.101,A -85,B 0,C 180,E1 -8531.914,E2 -8531.914} C_VEL
LIN {X 0,Y 452.808,Z 245.114,A -85,B 0,C 180,E1 -8534.7,E2 -8534.7} C_VEL
LIN {X 0,Y 452.821,Z 249.17,A -85,B 0,C 180,E1 -8538.284,E2 -8538.284} C_VEL
LIN {X 0,Y 456.165,Z 263.88,A -85,B 0,C 180,E1 -8538.867,E2 -8538.867} C_VEL
LIN {X 0,Y 456.566,Z 267.112,A -85,B 0,C 180,E1 -8539.017,E2 -8539.017} C_VEL
LIN {X 0,Y 456.325,Z 275.978,A -85,B 0,C 180,E1 -8539.443,E2 -8539.443} C_VEL
LIN {X 0,Y 455.477,Z 281.421,A -85,B 0,C 180,E1 -8539.733,E2 -8539.733} C_VEL
LIN {X 0,Y 450.88,Z 293.319,A -85,B 0,C 180,E1 -8540.429,E2 -8540.429} C_VEL
LIN {X 0,Y 448.622,Z 299.824,A -85,B 0,C 180,E1 -8540.92,E2 -8540.92} C_VEL
LIN {X 0,Y 448.121,Z 302.954,A -85,B 0,C 180,E1 -8541.208,E2 -8541.208} C_VEL
LIN {X 0,Y 447.669,Z 313.245,A -85,B 0,C 180,E1 -8542.33,E2 -8542.33} C_VEL
LIN {X 0,Y 447.163,Z 321.633,A -85,B 0,C 180,E1 -8543.456,E2 -8543.456} C_VEL
LIN {X 0,Y 446.627,Z 329.806,A -85,B 0,C 180,E1 -8544.807,E2 -8544.807} C_VEL
LIN {X 0,Y 446.248,Z 335.404,A -85,B 0,C 180,E1 -8545.935,E2 -8545.935} C_VEL
LIN {X 0,Y 445.807,Z 340.873,A -85,B 0,C 180,E1 -8547.288,E2 -8547.288} C_VEL
LIN {X 0,Y 445.7,Z 345.152,A -85,B 0,C 180,E1 -8548.643,E2 -8548.643} C_VEL
LIN {X 0,Y 445.475,Z 348.399,A -85,B 0,C 180,E1 -8549.999,E2 -8549.999} C_VEL
LIN {X 0,Y 445.526,Z 351.22,A -85,B 0,C 180,E1 -8551.807,E2 -8551.807} C_VEL
LIN {X 0,Y 445.555,Z 352.03,A -85,B 0,C 180,E1 -8552.711,E2 -8552.711} C_VEL
LIN {X 0,Y 445.584,Z 352.423,A -85,B 0,C 180,E1 -8553.616,E2 -8553.616} C_VEL
LIN {X 0,Y 445.533,Z 352.087,A -85,B 0,C 180,E1 -8555.43,E2 -8555.43} C_VEL
LIN {X 0,Y 445.578,Z 351.208,A -85,B 0,C 180,E1 -8556.44,E2 -8556.44} C_VEL
LIN {X 0,Y 445.665,Z 348.555,A -85,B 0,C 180,E1 -8558.158,E2 -8558.158} C_VEL
LIN {X 0,Y 445.834,Z 345.353,A -85,B 0,C 180,E1 -8559.526,E2 -8559.526} C_VEL
LIN {X 0,Y 446.051,Z 341.081,A -85,B 0,C 180,E1 -8560.897,E2 -8560.897} C_VEL
LIN {X 0,Y 446.398,Z 335.146,A -85,B 0,C 180,E1 -8562.376,E2 -8562.376} C_VEL
LIN {X 0,Y 446.903,Z 327.429,A -85,B 0,C 180,E1 -8563.875,E2 -8563.875} C_VEL
LIN {X 0,Y 447.503,Z 318.499,A -85,B 0,C 180,E1 -8565.25,E2 -8565.25} C_VEL
LIN {X 0,Y 448.115,Z 309.281,A -85,B 0,C 180,E1 -8566.396,E2 -8566.396} C_VEL
LIN {X 0,Y 448.622,Z 298.965,A -85,B 0,C 180,E1 -8567.433,E2 -8567.433} C_VEL
LIN {X 0,Y 449.291,Z 287.481,A -85,B 0,C 180,E1 -8568.347,E2 -8568.347} C_VEL
LIN {X 0,Y 449.703,Z 275.411,A -85,B 0,C 180,E1 -8569.098,E2 -8569.098} C_VEL
LIN {X 0,Y 449.945,Z 266.675,A -85,B 0,C 180,E1 -8569.515,E2 -8569.515} C_VEL
LIN {X 0,Y 446.891,Z 254.184,A -85,B 0,C 180,E1 -8570.094,E2 -8570.094} C_VEL
LIN {X 0,Y 445.67,Z 249.677,A -85,B 0,C 180,E1 -8570.278,E2 -8570.278} C_VEL
LIN {X 0,Y 445.74,Z 245.774,A -85,B 0,C 180,E1 -8573.866,E2 -8573.866} C_VEL
LIN {X 0,Y 445.802,Z 242.255,A -85,B 0,C 180,E1 -8577.204,E2 -8577.204} C_VEL
LIN {X 0,Y 445.871,Z 239.149,A -85,B 0,C 180,E1 -8580.29,E2 -8580.29} C_VEL
LIN {X 0,Y 445.942,Z 235.996,A -85,B 0,C 180,E1 -8583.475,E2 -8583.475} C_VEL
LIN {X 0,Y 446.055,Z 233.033,A -85,B 0,C 180,E1 -8586.529,E2 -8586.529} C_VEL
LIN {X 0,Y 446.351,Z 232.887,A -85,B 0,C 180,E1 -8589.508,E2 -8589.508} C_VEL
LIN {X 0,Y 446.423,Z 232.879,A -85,B 0,C 180,E1 -8592.603,E2 -8592.603} C_VEL
LIN {X 0,Y 446.446,Z 232.873,A -85,B 0,C 180,E1 -8595.102,E2 -8595.102} C_VEL
LIN {X 0,Y 446.41,Z 232.877,A -85,B 0,C 180,E1 -8598.607,E2 -8598.607} C_VEL
LIN {X 0,Y 446.433,Z 232.877,A -85,B 0,C 180,E1 -8600.971,E2 -8600.971} C_VEL
LIN {X 0,Y 446.412,Z 232.881,A -85,B 0,C 180,E1 -8604.373,E2 -8604.373} C_VEL
LIN {X 0,Y 446.411,Z 232.881,A -85,B 0,C 180,E1 -8607.637,E2 -8607.637} C_VEL
LIN {X 0,Y 446.439,Z 232.878,A -85,B 0,C 180,E1 -8610.79,E2 -8610.79} C_VEL
LIN {X 0,Y 446.468,Z 232.871,A -85,B 0,C 180,E1 -8613.848,E2 -8613.848} C_VEL
LIN {X 0,Y 446.419,Z 232.876,A -85,B 0,C 180,E1 -8616.823,E2 -8616.823} C_VEL
LIN {X 0,Y 446.433,Z 232.874,A -85,B 0,C 180,E1 -8619.736,E2 -8619.736} C_VEL
LIN {X 0,Y 446.451,Z 232.874,A -85,B 0,C 180,E1 -8622.596,E2 -8622.596} C_VEL
LIN {X 0,Y 446.459,Z 232.874,A -85,B 0,C 180,E1 -8625.412,E2 -8625.412} C_VEL
LIN {X 0,Y 446.505,Z 232.865,A -85,B 0,C 180,E1 -8628.193,E2 -8628.193} C_VEL
LIN {X 0,Y 446.588,Z 232.856,A -85,B 0,C 180,E1 -8631.857,E2 -8631.857} C_VEL
LIN {X 0,Y 446.644,Z 232.848,A -85,B 0,C 180,E1 -8634.582,E2 -8634.582} C_VEL
LIN {X 0,Y 446.699,Z 232.844,A -85,B 0,C 180,E1 -8637.295,E2 -8637.295} C_VEL
LIN {X 0,Y 446.778,Z 232.832,A -85,B 0,C 180,E1 -8640,E2 -8640} C_VEL
LIN {X 0,Y 446.698,Z 232.841,A -85,B 0,C 180,E1 -8642.705,E2 -8642.705} C_VEL
LIN {X 0,Y 446.641,Z 232.848,A -85,B 0,C 180,E1 -8646.324,E2 -8646.324} C_VEL
LIN {X 0,Y 446.525,Z 232.864,A -85,B 0,C 180,E1 -8649.056,E2 -8649.056} C_VEL
LIN {X 0,Y 446.509,Z 232.863,A -85,B 0,C 180,E1 -8652.73,E2 -8652.73} C_VEL
LIN {X 0,Y 446.485,Z 232.865,A -85,B 0,C 180,E1 -8656.228,E2 -8656.228} C_VEL
LIN {X 0,Y 446.458,Z 232.869,A -85,B 0,C 180,E1 -8659.304,E2 -8659.304} C_VEL
LIN {X 0,Y 446.406,Z 232.88,A -85,B 0,C 180,E1 -8662.2,E2 -8662.2} C_VEL
LIN {X 0,Y 446.447,Z 232.877,A -85,B 0,C 180,E1 -8665.153,E2 -8665.153} C_VEL
LIN {X 0,Y 446.474,Z 232.871,A -85,B 0,C 180,E1 -8668.179,E2 -8668.179} C_VEL
LIN {X 0,Y 446.409,Z 232.878,A -85,B 0,C 180,E1 -8671.301,E2 -8671.301} C_VEL
LIN {X 0,Y 446.419,Z 232.877,A -85,B 0,C 180,E1 -8674.524,E2 -8674.524} C_VEL
LIN {X 0,Y 446.407,Z 232.879,A -85,B 0,C 180,E1 -8678.08,E2 -8678.08} C_VEL
LIN {X 0,Y 446.414,Z 232.877,A -85,B 0,C 180,E1 -8680.918,E2 -8680.918} C_VEL
LIN {X 0,Y 446.392,Z 232.881,A -85,B 0,C 180,E1 -8683.847,E2 -8683.847} C_VEL
LIN {X 0,Y 446.392,Z 232.883,A -85,B 0,C 180,E1 -8686.404,E2 -8686.404} C_VEL
LIN {X 0,Y 446.44,Z 232.953,A -85,B 0,C 180,E1 -8688.16,E2 -8688.16} C_VEL
LIN {X 0,Y 447.522,Z 238.883,A -85,B 0,C 180,E1 -8691.087,E2 -8691.087} C_VEL
LIN {X 0,Y 448.341,Z 243.982,A -85,B 0,C 180,E1 -8693.441,E2 -8693.441} C_VEL
LIN {X 0,Y 448.276,Z 249.127,A -85,B 0,C 180,E1 -8695.641,E2 -8695.641} C_VEL
LIN {X 0,Y 447.755,Z 256.948,A -85,B 0,C 180,E1 -8698.806,E2 -8698.806} C_VEL
LIN {X 0,Y 447.263,Z 266.2,A -85,B 0,C 180,E1 -8702.386,E2 -8702.386} C_VEL
LIN {X 0,Y 446.835,Z 274.181,A -85,B 0,C 180,E1 -8705.369,E2 -8705.369} C_VEL
LIN {X 0,Y 446.505,Z 283.574,A -85,B 0,C 180,E1 -8708.777,E2 -8708.777} C_VEL
LIN {X 0,Y 446.203,Z 291.588,A -85,B 0,C 180,E1 -8711.64,E2 -8711.64} C_VEL
LIN {X 0,Y 446.003,Z 297.817,A -85,B 0,C 180,E1 -8713.82,E2 -8713.82} C_VEL
LIN {X 0,Y 448.377,Z 312.585,A -85,B 0,C 180,E1 -8714.327,E2 -8714.327} C_VEL
LIN {X 0,Y 449.376,Z 320.905,A -85,B 0,C 180,E1 -8714.699,E2 -8714.699} C_VEL
LIN {X 0,Y 448.932,Z 331.96,A -85,B 0,C 180,E1 -8715.264,E2 -8715.264} C_VEL
LIN {X 0,Y 448.323,Z 343.847,A -85,B 0,C 180,E1 -8716.055,E2 -8716.055} C_VEL
LIN {X 0,Y 447.741,Z 355.041,A -85,B 0,C 180,E1 -8717.012,E2 -8717.012} C_VEL
LIN {X 0,Y 447.288,Z 364.272,A -85,B 0,C 180,E1 -8717.985,E2 -8717.985} C_VEL
LIN {X 0,Y 446.713,Z 373.162,A -85,B 0,C 180,E1 -8719.119,E2 -8719.119} C_VEL
LIN {X 0,Y 446.256,Z 381.843,A -85,B 0,C 180,E1 -8720.483,E2 -8720.483} C_VEL
LIN {X 0,Y 445.883,Z 388.785,A -85,B 0,C 180,E1 -8721.846,E2 -8721.846} C_VEL
LIN {X 0,Y 445.648,Z 394.356,A -85,B 0,C 180,E1 -8723.209,E2 -8723.209} C_VEL
LIN {X 0,Y 445.54,Z 398.728,A -85,B 0,C 180,E1 -8724.57,E2 -8724.57} C_VEL
LIN {X 0,Y 445.427,Z 401.04,A -85,B 0,C 180,E1 -8725.477,E2 -8725.477} C_VEL
LIN {X 0,Y 445.397,Z 402.918,A -85,B 0,C 180,E1 -8726.383,E2 -8726.383} C_VEL
LIN {X 0,Y 445.422,Z 404.329,A -85,B 0,C 180,E1 -8727.288,E2 -8727.288} C_VEL
LIN {X 0,Y 445.372,Z 405.946,A -85,B 0,C 180,E1 -8729.097,E2 -8729.097} C_VEL
LIN {X 0,Y 445.349,Z 406.163,A -85,B 0,C 180,E1 -8730.001,E2 -8730.001} C_VEL
LIN {X 0,Y 445.372,Z 405.946,A -85,B 0,C 180,E1 -8730.905,E2 -8730.905} C_VEL
LIN {X 0,Y 445.423,Z 404.332,A -85,B 0,C 180,E1 -8732.714,E2 -8732.714} C_VEL
LIN {X 0,Y 445.398,Z 402.921,A -85,B 0,C 180,E1 -8733.62,E2 -8733.62} C_VEL
LIN {X 0,Y 445.501,Z 399.964,A -85,B 0,C 180,E1 -8734.979,E2 -8734.979} C_VEL
LIN {X 0,Y 445.588,Z 395.579,A -85,B 0,C 180,E1 -8736.452,E2 -8736.452} C_VEL
LIN {X 0,Y 445.806,Z 389.801,A -85,B 0,C 180,E1 -8737.93,E2 -8737.93} C_VEL
LIN {X 0,Y 446.187,Z 383.086,A -85,B 0,C 180,E1 -8739.292,E2 -8739.292} C_VEL
LIN {X 0,Y 446.635,Z 374.755,A -85,B 0,C 180,E1 -8740.656,E2 -8740.656} C_VEL
LIN {X 0,Y 447.171,Z 366.226,A -85,B 0,C 180,E1 -8741.791,E2 -8741.791} C_VEL
LIN {X 0,Y 447.704,Z 356.472,A -85,B 0,C 180,E1 -8742.851,E2 -8742.851} C_VEL
LIN {X 0,Y 448.255,Z 345.272,A -85,B 0,C 180,E1 -8743.835,E2 -8743.835} C_VEL
LIN {X 0,Y 448.841,Z 333.864,A -85,B 0,C 180,E1 -8744.626,E2 -8744.626} C_VEL
LIN {X 0,Y 449.373,Z 322.165,A -85,B 0,C 180,E1 -8745.246,E2 -8745.246} C_VEL
LIN {X 0,Y 449.013,Z 316.699,A -85,B 0,C 180,E1 -8745.496,E2 -8745.496} C_VEL
LIN {X 0,Y 446.842,Z 303.128,A -85,B 0,C 180,E1 -8746.013,E2 -8746.013} C_VEL
LIN {X 0,Y 446.011,Z 297.827,A -85,B 0,C 180,E1 -8746.185,E2 -8746.185} C_VEL
LIN {X 0,Y 446.33,Z 288.948,A -85,B 0,C 180,E1 -8749.311,E2 -8749.311} C_VEL
LIN {X 0,Y 446.645,Z 279.581,A -85,B 0,C 180,E1 -8752.677,E2 -8752.677} C_VEL
LIN {X 0,Y 447.104,Z 269.51,A -85,B 0,C 180,E1 -8756.365,E2 -8756.365} C_VEL
LIN {X 0,Y 447.403,Z 262.134,A -85,B 0,C 180,E1 -8759.142,E2 -8759.142} C_VEL
LIN {X 0,Y 447.914,Z 254.094,A -85,B 0,C 180,E1 -8762.242,E2 -8762.242} C_VEL
LIN {X 0,Y 448.34,Z 246.102,A -85,B 0,C 180,E1 -8765.452,E2 -8765.452} C_VEL
LIN {X 0,Y 448.162,Z 242.71,A -85,B 0,C 180,E1 -8766.891,E2 -8766.891} C_VEL
LIN {X 0,Y 447.13,Z 236.635,A -85,B 0,C 180,E1 -8769.63,E2 -8769.63} C_VEL
LIN {X 0,Y 446.456,Z 232.876,A -85,B 0,C 180,E1 -8771.464,E2 -8771.464} C_VEL
LIN {X 0,Y 446.46,Z 232.875,A -85,B 0,C 180,E1 -8775.104,E2 -8775.104} C_VEL
LIN {X 0,Y 446.435,Z 232.875,A -85,B 0,C 180,E1 -8778.61,E2 -8778.61} C_VEL
LIN {X 0,Y 446.447,Z 232.876,A -85,B 0,C 180,E1 -8780.973,E2 -8780.973} C_VEL
LIN {X 0,Y 446.421,Z 232.878,A -85,B 0,C 180,E1 -8784.374,E2 -8784.374} C_VEL
LIN {X 0,Y 446.422,Z 232.874,A -85,B 0,C 180,E1 -8787.638,E2 -8787.638} C_VEL
LIN {X 0,Y 446.443,Z 232.874,A -85,B 0,C 180,E1 -8790.79,E2 -8790.79} C_VEL
LIN {X 0,Y 446.447,Z 232.875,A -85,B 0,C 180,E1 -8793.846,E2 -8793.846} C_VEL
LIN {X 0,Y 446.433,Z 232.876,A -85,B 0,C 180,E1 -8796.824,E2 -8796.824} C_VEL
LIN {X 0,Y 446.45,Z 232.873,A -85,B 0,C 180,E1 -8799.737,E2 -8799.737} C_VEL
LIN {X 0,Y 446.443,Z 232.874,A -85,B 0,C 180,E1 -8802.596,E2 -8802.596} C_VEL
LIN {X 0,Y 446.46,Z 232.87,A -85,B 0,C 180,E1 -8805.412,E2 -8805.412} C_VEL
LIN {X 0,Y 446.512,Z 232.865,A -85,B 0,C 180,E1 -8808.193,E2 -8808.193} C_VEL
LIN {X 0,Y 446.526,Z 232.863,A -85,B 0,C 180,E1 -8810.944,E2 -8810.944} C_VEL
LIN {X 0,Y 446.642,Z 232.85,A -85,B 0,C 180,E1 -8813.676,E2 -8813.676} C_VEL
LIN {X 0,Y 446.697,Z 232.843,A -85,B 0,C 180,E1 -8817.295,E2 -8817.295} C_VEL
LIN {X 0,Y 446.797,Z 232.831,A -85,B 0,C 180,E1 -8820,E2 -8820} C_VEL
LIN {X 0,Y 446.686,Z 232.843,A -85,B 0,C 180,E1 -8822.706,E2 -8822.706} C_VEL
LIN {X 0,Y 446.605,Z 232.85,A -85,B 0,C 180,E1 -8826.324,E2 -8826.324} C_VEL
LIN {X 0,Y 446.528,Z 232.866,A -85,B 0,C 180,E1 -8829.056,E2 -8829.056} C_VEL
LIN {X 0,Y 446.53,Z 232.865,A -85,B 0,C 180,E1 -8832.73,E2 -8832.73} C_VEL
LIN {X 0,Y 446.497,Z 232.868,A -85,B 0,C 180,E1 -8836.459,E2 -8836.459} C_VEL
LIN {X 0,Y 446.476,Z 232.873,A -85,B 0,C 180,E1 -8839.303,E2 -8839.303} C_VEL
LIN {X 0,Y 446.424,Z 232.876,A -85,B 0,C 180,E1 -8842.2,E2 -8842.2} C_VEL
LIN {X 0,Y 446.419,Z 232.877,A -85,B 0,C 180,E1 -8845.155,E2 -8845.155} C_VEL
LIN {X 0,Y 446.423,Z 232.875,A -85,B 0,C 180,E1 -8848.183,E2 -8848.183} C_VEL
LIN {X 0,Y 446.422,Z 232.876,A -85,B 0,C 180,E1 -8851.3,E2 -8851.3} C_VEL
LIN {X 0,Y 446.43,Z 232.876,A -85,B 0,C 180,E1 -8854.523,E2 -8854.523} C_VEL
LIN {X 0,Y 446.418,Z 232.878,A -85,B 0,C 180,E1 -8858.078,E2 -8858.078} C_VEL
LIN {X 0,Y 446.429,Z 232.876,A -85,B 0,C 180,E1 -8860.916,E2 -8860.916} C_VEL
LIN {X 0,Y 446.405,Z 232.878,A -85,B 0,C 180,E1 -8863.846,E2 -8863.846} C_VEL
LIN {X 0,Y 446.389,Z 232.882,A -85,B 0,C 180,E1 -8866.405,E2 -8866.405} C_VEL
LIN {X 0,Y 446.4,Z 232.881,A -85,B 0,C 180,E1 -8869.796,E2 -8869.796} C_VEL
LIN {X 0,Y 446.41,Z 232.879,A -85,B 0,C 180,E1 -8872.12,E2 -8872.12} C_VEL
LIN {X 0,Y 446.428,Z 232.878,A -85,B 0,C 180,E1 -8875.476,E2 -8875.476} C_VEL
LIN {X 0,Y 446.348,Z 232.888,A -85,B 0,C 180,E1 -8878.241,E2 -8878.241} C_VEL
LIN {X 0,Y 446.13,Z 232.913,A -85,B 0,C 180,E1 -8880.766,E2 -8880.766} C_VEL
LIN {X 0,Y 445.958,Z 232.938,A -85,B 0,C 180,E1 -8881.949,E2 -8881.949} C_VEL
LIN {X 0,Y 445.87,Z 234.469,A -85,B 0,C 180,E1 -8883.809,E2 -8883.809} C_VEL
LIN {X 0,Y 445.816,Z 237.489,A -85,B 0,C 180,E1 -8886.788,E2 -8886.788} C_VEL
LIN {X 0,Y 445.749,Z 240.487,A -85,B 0,C 180,E1 -8889.703,E2 -8889.703} C_VEL
LIN {X 0,Y 445.723,Z 243.511,A -85,B 0,C 180,E1 -8892.566,E2 -8892.566} C_VEL
LIN {X 0,Y 445.69,Z 246.561,A -85,B 0,C 180,E1 -8895.385,E2 -8895.385} C_VEL
LIN {X 0,Y 445.803,Z 249.767,A -85,B 0,C 180,E1 -8898.06,E2 -8898.06} C_VEL
LIN {X 0,Y 448.839,Z 263.034,A -85,B 0,C 180,E1 -8898.583,E2 -8898.583} C_VEL
LIN {X 0,Y 449.694,Z 267.318,A -85,B 0,C 180,E1 -8898.79,E2 -8898.79} C_VEL
LIN {X 0,Y 449.297,Z 279.507,A -85,B 0,C 180,E1 -8899.408,E2 -8899.408} C_VEL
LIN {X 0,Y 448.765,Z 291.243,A -85,B 0,C 180,E1 -8900.193,E2 -8900.193} C_VEL
LIN {X 0,Y 448.121,Z 302.954,A -85,B 0,C 180,E1 -8901.208,E2 -8901.208} C_VEL
LIN {X 0,Y 447.238,Z 307.613,A -85,B 0,C 180,E1 -8901.66,E2 -8901.66} C_VEL
LIN {X 0,Y 444.173,Z 314.948,A -85,B 0,C 180,E1 -8902.421,E2 -8902.421} C_VEL
LIN {X 0,Y 441.012,Z 321.715,A -85,B 0,C 180,E1 -8903.265,E2 -8903.265} C_VEL
LIN {X 0,Y 439.99,Z 325.483,A -85,B 0,C 180,E1 -8903.843,E2 -8903.843} C_VEL
LIN {X 0,Y 439.456,Z 332.832,A -85,B 0,C 180,E1 -8905.182,E2 -8905.182} C_VEL
LIN {X 0,Y 438.929,Z 339.795,A -85,B 0,C 180,E1 -8906.786,E2 -8906.786} C_VEL
LIN {X 0,Y 438.589,Z 344.428,A -85,B 0,C 180,E1 -8908.162,E2 -8908.162} C_VEL
LIN {X 0,Y 438.516,Z 347.96,A -85,B 0,C 180,E1 -8909.54,E2 -8909.54} C_VEL
LIN {X 0,Y 438.396,Z 350.508,A -85,B 0,C 180,E1 -8910.917,E2 -8910.917} C_VEL
LIN {X 0,Y 438.469,Z 351.703,A -85,B 0,C 180,E1 -8911.836,E2 -8911.836} C_VEL
LIN {X 0,Y 438.48,Z 352.481,A -85,B 0,C 180,E1 -8912.755,E2 -8912.755} C_VEL
LIN {X 0,Y 438.497,Z 352.858,A -85,B 0,C 180,E1 -8913.674,E2 -8913.674} C_VEL
LIN {X 0,Y 438.474,Z 352.488,A -85,B 0,C 180,E1 -8915.517,E2 -8915.517} C_VEL
LIN {X 0,Y 438.506,Z 351.702,A -85,B 0,C 180,E1 -8916.44,E2 -8916.44} C_VEL
LIN {X 0,Y 438.559,Z 350.495,A -85,B 0,C 180,E1 -8917.364,E2 -8917.364} C_VEL
LIN {X 0,Y 438.667,Z 347.927,A -85,B 0,C 180,E1 -8918.753,E2 -8918.753} C_VEL
LIN {X 0,Y 438.818,Z 344.349,A -85,B 0,C 180,E1 -8920.145,E2 -8920.145} C_VEL
LIN {X 0,Y 439.151,Z 339.647,A -85,B 0,C 180,E1 -8921.538,E2 -8921.538} C_VEL
LIN {X 0,Y 439.602,Z 332.569,A -85,B 0,C 180,E1 -8923.167,E2 -8923.167} C_VEL
LIN {X 0,Y 440.147,Z 324.817,A -85,B 0,C 180,E1 -8924.564,E2 -8924.564} C_VEL
LIN {X 0,Y 440.827,Z 315.084,A -85,B 0,C 180,E1 -8925.961,E2 -8925.961} C_VEL
LIN {X 0,Y 441.464,Z 304.986,A -85,B 0,C 180,E1 -8927.123,E2 -8927.123} C_VEL
LIN {X 0,Y 442.068,Z 294.839,A -85,B 0,C 180,E1 -8928.058,E2 -8928.058} C_VEL
LIN {X 0,Y 442.674,Z 283.797,A -85,B 0,C 180,E1 -8928.872,E2 -8928.872} C_VEL
LIN {X 0,Y 443.067,Z 272.374,A -85,B 0,C 180,E1 -8929.53,E2 -8929.53} C_VEL
LIN {X 0,Y 443.214,Z 268.42,A -85,B 0,C 180,E1 -8929.715,E2 -8929.715} C_VEL
LIN {X 0,Y 440.318,Z 256.42,A -85,B 0,C 180,E1 -8930.302,E2 -8930.302} C_VEL
LIN {X 0,Y 438.592,Z 250.099,A -85,B 0,C 180,E1 -8930.564,E2 -8930.564} C_VEL
LIN {X 0,Y 438.695,Z 246.329,A -85,B 0,C 180,E1 -8934.054,E2 -8934.054} C_VEL
LIN {X 0,Y 438.743,Z 243.616,A -85,B 0,C 180,E1 -8936.647,E2 -8936.647} C_VEL
LIN {X 0,Y 438.821,Z 240.458,A -85,B 0,C 180,E1 -8939.766,E2 -8939.766} C_VEL
LIN {X 0,Y 438.86,Z 237.278,A -85,B 0,C 180,E1 -8942.988,E2 -8942.988} C_VEL
LIN {X 0,Y 438.988,Z 234.084,A -85,B 0,C 180,E1 -8946.322,E2 -8946.322} C_VEL
LIN {X 0,Y 439.096,Z 233.793,A -85,B 0,C 180,E1 -8947.458,E2 -8947.458} C_VEL
LIN {X 0,Y 439.313,Z 233.762,A -85,B 0,C 180,E1 -8949.835,E2 -8949.835} C_VEL
LIN {X 0,Y 439.375,Z 233.757,A -85,B 0,C 180,E1 -8952.626,E2 -8952.626} C_VEL
LIN {X 0,Y 439.394,Z 233.752,A -85,B 0,C 180,E1 -8955.269,E2 -8955.269} C_VEL
LIN {X 0,Y 439.373,Z 233.755,A -85,B 0,C 180,E1 -8958.743,E2 -8958.743} C_VEL
LIN {X 0,Y 439.373,Z 233.754,A -85,B 0,C 180,E1 -8961.605,E2 -8961.605} C_VEL
LIN {X 0,Y 439.392,Z 233.752,A -85,B 0,C 180,E1 -8964.843,E2 -8964.843} C_VEL
LIN {X 0,Y 439.362,Z 233.755,A -85,B 0,C 180,E1 -8968.138,E2 -8968.138} C_VEL
LIN {X 0,Y 439.423,Z 233.747,A -85,B 0,C 180,E1 -8971.597,E2 -8971.597} C_VEL
LIN {X 0,Y 439.396,Z 233.753,A -85,B 0,C 180,E1 -8974.414,E2 -8974.414} C_VEL
LIN {X 0,Y 439.355,Z 233.76,A -85,B 0,C 180,E1 -8977.424,E2 -8977.424} C_VEL
LIN {X 0,Y 439.43,Z 233.751,A -85,B 0,C 180,E1 -8980.662,E2 -8980.662} C_VEL
LIN {X 0,Y 439.451,Z 233.747,A -85,B 0,C 180,E1 -8984.224,E2 -8984.224} C_VEL
LIN {X 0,Y 439.471,Z 233.741,A -85,B 0,C 180,E1 -8988.001,E2 -8988.001} C_VEL
LIN {X 0,Y 439.536,Z 233.734,A -85,B 0,C 180,E1 -8991.726,E2 -8991.726} C_VEL
LIN {X 0,Y 439.618,Z 233.724,A -85,B 0,C 180,E1 -8994.496,E2 -8994.496} C_VEL
LIN {X 0,Y 439.625,Z 233.722,A -85,B 0,C 180,E1 -8998.168,E2 -8998.168} C_VEL
LIN {X 0,Y 439.748,Z 233.708,A -85,B 0,C 180,E1 -9000,E2 -9000} C_VEL
LIN {X 0,Y 439.645,Z 233.72,A -85,B 0,C 180,E1 -9002.749,E2 -9002.749} C_VEL
LIN {X 0,Y 439.611,Z 233.724,A -85,B 0,C 180,E1 -9006.425,E2 -9006.425} C_VEL
LIN {X 0,Y 439.487,Z 233.74,A -85,B 0,C 180,E1 -9009.202,E2 -9009.202} C_VEL
LIN {X 0,Y 439.453,Z 233.742,A -85,B 0,C 180,E1 -9012.938,E2 -9012.938} C_VEL
LIN {X 0,Y 439.436,Z 233.744,A -85,B 0,C 180,E1 -9016.349,E2 -9016.349} C_VEL
LIN {X 0,Y 439.391,Z 233.749,A -85,B 0,C 180,E1 -9019.627,E2 -9019.627} C_VEL
LIN {X 0,Y 439.353,Z 233.756,A -85,B 0,C 180,E1 -9022.576,E2 -9022.576} C_VEL
LIN {X 0,Y 439.394,Z 233.752,A -85,B 0,C 180,E1 -9025.586,E2 -9025.586} C_VEL
LIN {X 0,Y 439.415,Z 233.752,A -85,B 0,C 180,E1 -9028.674,E2 -9028.674} C_VEL
LIN {X 0,Y 439.372,Z 233.756,A -85,B 0,C 180,E1 -9032.034,E2 -9032.034} C_VEL
LIN {X 0,Y 439.385,Z 233.753,A -85,B 0,C 180,E1 -9035.341,E2 -9035.341} C_VEL
LIN {X 0,Y 439.37,Z 233.757,A -85,B 0,C 180,E1 -9038.596,E2 -9038.596} C_VEL
LIN {X 0,Y 439.374,Z 233.755,A -85,B 0,C 180,E1 -9041.257,E2 -9041.257} C_VEL
LIN {X 0,Y 439.393,Z 233.756,A -85,B 0,C 180,E1 -9044.73,E2 -9044.73} C_VEL
LIN {X 0,Y 439.418,Z 233.839,A -85,B 0,C 180,E1 -9047.8,E2 -9047.8} C_VEL
LIN {X 0,Y 440.546,Z 240.019,A -85,B 0,C 180,E1 -9050.915,E2 -9050.915} C_VEL
LIN {X 0,Y 441.38,Z 245.197,A -85,B 0,C 180,E1 -9053.36,E2 -9053.36} C_VEL
LIN {X 0,Y 441.306,Z 250.158,A -85,B 0,C 180,E1 -9055.522,E2 -9055.522} C_VEL
LIN {X 0,Y 440.841,Z 256.776,A -85,B 0,C 180,E1 -9058.26,E2 -9058.26} C_VEL
LIN {X 0,Y 440.311,Z 265.978,A -85,B 0,C 180,E1 -9061.911,E2 -9061.911} C_VEL
LIN {X 0,Y 439.855,Z 273.917,A -85,B 0,C 180,E1 -9064.951,E2 -9064.951} C_VEL
LIN {X 0,Y 439.449,Z 283.222,A -85,B 0,C 180,E1 -9068.42,E2 -9068.42} C_VEL
LIN {X 0,Y 439.146,Z 291.232,A -85,B 0,C 180,E1 -9071.334,E2 -9071.334} C_VEL
LIN {X 0,Y 438.918,Z 297.617,A -85,B 0,C 180,E1 -9073.575,E2 -9073.575} C_VEL
LIN {X 0,Y 441.113,Z 311.059,A -85,B 0,C 180,E1 -9074.023,E2 -9074.023} C_VEL
LIN {X 0,Y 442.475,Z 320.47,A -85,B 0,C 180,E1 -9074.454,E2 -9074.454} C_VEL
LIN {X 0,Y 442.048,Z 331.527,A -85,B 0,C 180,E1 -9075.029,E2 -9075.029} C_VEL
LIN {X 0,Y 441.392,Z 343.413,A -85,B 0,C 180,E1 -9075.831,E2 -9075.831} C_VEL
LIN {X 0,Y 440.745,Z 355.111,A -85,B 0,C 180,E1 -9076.853,E2 -9076.853} C_VEL
LIN {X 0,Y 440.191,Z 365.797,A -85,B 0,C 180,E1 -9078.022,E2 -9078.022} C_VEL
LIN {X 0,Y 439.619,Z 374.324,A -85,B 0,C 180,E1 -9079.175,E2 -9079.175} C_VEL
LIN {X 0,Y 439.15,Z 382.655,A -85,B 0,C 180,E1 -9080.56,E2 -9080.56} C_VEL
LIN {X 0,Y 438.75,Z 389.371,A -85,B 0,C 180,E1 -9081.944,E2 -9081.944} C_VEL
LIN {X 0,Y 438.524,Z 395.529,A -85,B 0,C 180,E1 -9083.56,E2 -9083.56} C_VEL
LIN {X 0,Y 438.434,Z 399.534,A -85,B 0,C 180,E1 -9084.943,E2 -9084.943} C_VEL
LIN {X 0,Y 438.302,Z 402.488,A -85,B 0,C 180,E1 -9086.324,E2 -9086.324} C_VEL
LIN {X 0,Y 438.35,Z 403.902,A -85,B 0,C 180,E1 -9087.244,E2 -9087.244} C_VEL
LIN {X 0,Y 438.283,Z 405.519,A -85,B 0,C 180,E1 -9089.083,E2 -9089.083} C_VEL
LIN {X 0,Y 438.29,Z 405.738,A -85,B 0,C 180,E1 -9090.001,E2 -9090.001} C_VEL
LIN {X 0,Y 438.283,Z 405.519,A -85,B 0,C 180,E1 -9090.92,E2 -9090.92} C_VEL
LIN {X 0,Y 438.351,Z 403.906,A -85,B 0,C 180,E1 -9092.758,E2 -9092.758} C_VEL
LIN {X 0,Y 438.303,Z 402.494,A -85,B 0,C 180,E1 -9093.679,E2 -9093.679} C_VEL
LIN {X 0,Y 438.435,Z 399.538,A -85,B 0,C 180,E1 -9095.059,E2 -9095.059} C_VEL
LIN {X 0,Y 438.507,Z 395.53,A -85,B 0,C 180,E1 -9096.443,E2 -9096.443} C_VEL
LIN {X 0,Y 438.754,Z 389.374,A -85,B 0,C 180,E1 -9098.058,E2 -9098.058} C_VEL
LIN {X 0,Y 439.153,Z 382.658,A -85,B 0,C 180,E1 -9099.443,E2 -9099.443} C_VEL
LIN {X 0,Y 439.622,Z 374.328,A -85,B 0,C 180,E1 -9100.828,E2 -9100.828} C_VEL
LIN {X 0,Y 440.193,Z 365.799,A -85,B 0,C 180,E1 -9101.98,E2 -9101.98} C_VEL
LIN {X 0,Y 440.732,Z 356.269,A -85,B 0,C 180,E1 -9103.036,E2 -9103.036} C_VEL
LIN {X 0,Y 441.339,Z 344.846,A -85,B 0,C 180,E1 -9104.056,E2 -9104.056} C_VEL
LIN {X 0,Y 441.938,Z 333.436,A -85,B 0,C 180,E1 -9104.86,E2 -9104.86} C_VEL
LIN {X 0,Y 442.499,Z 321.738,A -85,B 0,C 180,E1 -9105.489,E2 -9105.489} C_VEL
LIN {X 0,Y 441.08,Z 310.88,A -85,B 0,C 180,E1 -9105.985,E2 -9105.985} C_VEL
LIN {X 0,Y 438.912,Z 297.388,A -85,B 0,C 180,E1 -9106.453,E2 -9106.453} C_VEL
LIN {X 0,Y 439.263,Z 288.598,A -85,B 0,C 180,E1 -9109.634,E2 -9109.634} C_VEL
LIN {X 0,Y 439.554,Z 280.602,A -85,B 0,C 180,E1 -9112.566,E2 -9112.566} C_VEL
LIN {X 0,Y 440.02,Z 271.237,A -85,B 0,C 180,E1 -9116.056,E2 -9116.056} C_VEL
LIN {X 0,Y 440.346,Z 264.478,A -85,B 0,C 180,E1 -9118.621,E2 -9118.621} C_VEL
LIN {X 0,Y 440.824,Z 256.475,A -85,B 0,C 180,E1 -9121.745,E2 -9121.745} C_VEL
LIN {X 0,Y 441.306,Z 248.5,A -85,B 0,C 180,E1 -9124.983,E2 -9124.983} C_VEL
LIN {X 0,Y 441.272,Z 244.603,A -85,B 0,C 180,E1 -9126.636,E2 -9126.636} C_VEL
LIN {X 0,Y 440.146,Z 237.915,A -85,B 0,C 180,E1 -9129.696,E2 -9129.696} C_VEL
LIN {X 0,Y 439.424,Z 233.752,A -85,B 0,C 180,E1 -9131.761,E2 -9131.761} C_VEL
LIN {X 0,Y 439.408,Z 233.755,A -85,B 0,C 180,E1 -9135.272,E2 -9135.272} C_VEL
LIN {X 0,Y 439.395,Z 233.753,A -85,B 0,C 180,E1 -9138.744,E2 -9138.744} C_VEL
LIN {X 0,Y 439.378,Z 233.752,A -85,B 0,C 180,E1 -9141.609,E2 -9141.609} C_VEL
LIN {X 0,Y 439.4,Z 233.752,A -85,B 0,C 180,E1 -9144.844,E2 -9144.844} C_VEL
LIN {X 0,Y 439.375,Z 233.755,A -85,B 0,C 180,E1 -9148.14,E2 -9148.14} C_VEL
LIN {X 0,Y 439.416,Z 233.749,A -85,B 0,C 180,E1 -9151.604,E2 -9151.604} C_VEL
LIN {X 0,Y 439.387,Z 233.754,A -85,B 0,C 180,E1 -9154.414,E2 -9154.414} C_VEL
LIN {X 0,Y 439.371,Z 233.755,A -85,B 0,C 180,E1 -9157.425,E2 -9157.425} C_VEL
LIN {X 0,Y 439.448,Z 233.746,A -85,B 0,C 180,E1 -9160.664,E2 -9160.664} C_VEL
LIN {X 0,Y 439.425,Z 233.75,A -85,B 0,C 180,E1 -9164.223,E2 -9164.223} C_VEL
LIN {X 0,Y 439.491,Z 233.738,A -85,B 0,C 180,E1 -9167.286,E2 -9167.286} C_VEL
LIN {X 0,Y 439.489,Z 233.739,A -85,B 0,C 180,E1 -9170.798,E2 -9170.798} C_VEL
LIN {X 0,Y 439.612,Z 233.727,A -85,B 0,C 180,E1 -9173.575,E2 -9173.575} C_VEL
LIN {X 0,Y 439.646,Z 233.722,A -85,B 0,C 180,E1 -9177.251,E2 -9177.251} C_VEL
LIN {X 0,Y 439.766,Z 233.707,A -85,B 0,C 180,E1 -9180,E2 -9180} C_VEL
LIN {X 0,Y 439.635,Z 233.721,A -85,B 0,C 180,E1 -9182.749,E2 -9182.749} C_VEL
LIN {X 0,Y 439.557,Z 233.729,A -85,B 0,C 180,E1 -9186.426,E2 -9186.426} C_VEL
LIN {X 0,Y 439.492,Z 233.743,A -85,B 0,C 180,E1 -9189.202,E2 -9189.202} C_VEL
LIN {X 0,Y 439.474,Z 233.745,A -85,B 0,C 180,E1 -9192.938,E2 -9192.938} C_VEL
LIN {X 0,Y 439.455,Z 233.745,A -85,B 0,C 180,E1 -9196.348,E2 -9196.348} C_VEL
LIN {X 0,Y 439.41,Z 233.75,A -85,B 0,C 180,E1 -9199.626,E2 -9199.626} C_VEL
LIN {X 0,Y 439.369,Z 233.755,A -85,B 0,C 180,E1 -9202.575,E2 -9202.575} C_VEL
LIN {X 0,Y 439.36,Z 233.754,A -85,B 0,C 180,E1 -9205.588,E2 -9205.588} C_VEL
LIN {X 0,Y 439.389,Z 233.756,A -85,B 0,C 180,E1 -9208.676,E2 -9208.676} C_VEL
LIN {X 0,Y 439.376,Z 233.755,A -85,B 0,C 180,E1 -9212.03,E2 -9212.03} C_VEL
LIN {X 0,Y 439.398,Z 233.751,A -85,B 0,C 180,E1 -9215.339,E2 -9215.339} C_VEL
LIN {X 0,Y 439.376,Z 233.756,A -85,B 0,C 180,E1 -9218.596,E2 -9218.596} C_VEL
LIN {X 0,Y 439.388,Z 233.752,A -85,B 0,C 180,E1 -9221.255,E2 -9221.255} C_VEL
LIN {X 0,Y 439.383,Z 233.753,A -85,B 0,C 180,E1 -9224.732,E2 -9224.732} C_VEL
LIN {X 0,Y 439.351,Z 233.757,A -85,B 0,C 180,E1 -9227.789,E2 -9227.789} C_VEL
LIN {X 0,Y 439.365,Z 233.755,A -85,B 0,C 180,E1 -9231.402,E2 -9231.402} C_VEL
LIN {X 0,Y 439.402,Z 233.75,A -85,B 0,C 180,E1 -9234.843,E2 -9234.843} C_VEL
LIN {X 0,Y 439.312,Z 233.764,A -85,B 0,C 180,E1 -9238.133,E2 -9238.133} C_VEL
LIN {X 0,Y 438.999,Z 233.804,A -85,B 0,C 180,E1 -9241.295,E2 -9241.295} C_VEL
LIN {X 0,Y 438.854,Z 233.823,A -85,B 0,C 180,E1 -9242.326,E2 -9242.326} C_VEL
LIN {X 0,Y 438.796,Z 236.806,A -85,B 0,C 180,E1 -9245.389,E2 -9245.389} C_VEL
LIN {X 0,Y 438.73,Z 239.847,A -85,B 0,C 180,E1 -9248.38,E2 -9248.38} C_VEL
LIN {X 0,Y 438.69,Z 242.88,A -85,B 0,C 180,E1 -9251.311,E2 -9251.311} C_VEL
LIN {X 0,Y 438.695,Z 245.95,A -85,B 0,C 180,E1 -9254.195,E2 -9254.195} C_VEL
LIN {X 0,Y 438.69,Z 250.162,A -85,B 0,C 180,E1 -9257.813,E2 -9257.813} C_VEL
LIN {X 0,Y 441.783,Z 263.225,A -85,B 0,C 180,E1 -9258.34,E2 -9258.34} C_VEL
LIN {X 0,Y 442.788,Z 268.793,A -85,B 0,C 180,E1 -9258.613,E2 -9258.613} C_VEL
LIN {X 0,Y 442.384,Z 280.734,A -85,B 0,C 180,E1 -9259.24,E2 -9259.24} C_VEL
LIN {X 0,Y 441.831,Z 292.244,A -85,B 0,C 180,E1 -9260.037,E2 -9260.037} C_VEL
LIN {X 0,Y 441.166,Z 304.032,A -85,B 0,C 180,E1 -9261.086,E2 -9261.086} C_VEL
LIN {X 0,Y 440.699,Z 314.048,A -85,B 0,C 180,E1 -9262.208,E2 -9262.208} C_VEL
LIN {X 0,Y 440.054,Z 323.827,A -85,B 0,C 180,E1 -9263.58,E2 -9263.58} C_VEL
LIN {X 0,Y 439.99,Z 325.483,A -85,B 0,C 180,E1 -9263.843,E2 -9263.843} C_VEL
LIN {X 0,Y 438.952,Z 329.127,A -85,B 0,C 180,E1 -9264.446,E2 -9264.446} C_VEL
LIN {X 0,Y 434.316,Z 336.629,A -85,B 0,C 180,E1 -9265.855,E2 -9265.855} C_VEL
LIN {X 0,Y 432.161,Z 340.356,A -85,B 0,C 180,E1 -9266.73,E2 -9266.73} C_VEL
LIN {X 0,Y 431.713,Z 342.032,A -85,B 0,C 180,E1 -9267.194,E2 -9267.194} C_VEL
LIN {X 0,Y 431.539,Z 346.258,A -85,B 0,C 180,E1 -9268.599,E2 -9268.599} C_VEL
LIN {X 0,Y 431.344,Z 349.432,A -85,B 0,C 180,E1 -9269.999,E2 -9269.999} C_VEL
LIN {X 0,Y 431.382,Z 352.184,A -85,B 0,C 180,E1 -9271.866,E2 -9271.866} C_VEL
LIN {X 0,Y 431.406,Z 352.932,A -85,B 0,C 180,E1 -9272.8,E2 -9272.8} C_VEL
LIN {X 0,Y 431.413,Z 353.294,A -85,B 0,C 180,E1 -9273.735,E2 -9273.735} C_VEL
LIN {X 0,Y 431.416,Z 352.89,A -85,B 0,C 180,E1 -9275.608,E2 -9275.608} C_VEL
LIN {X 0,Y 431.438,Z 352.072,A -85,B 0,C 180,E1 -9276.546,E2 -9276.546} C_VEL
LIN {X 0,Y 431.559,Z 349.229,A -85,B 0,C 180,E1 -9278.427,E2 -9278.427} C_VEL
LIN {X 0,Y 431.734,Z 345.958,A -85,B 0,C 180,E1 -9279.84,E2 -9279.84} C_VEL
LIN {X 0,Y 432.047,Z 341.608,A -85,B 0,C 180,E1 -9281.255,E2 -9281.255} C_VEL
LIN {X 0,Y 432.456,Z 335.436,A -85,B 0,C 180,E1 -9282.816,E2 -9282.816} C_VEL
LIN {X 0,Y 433.034,Z 327.735,A -85,B 0,C 180,E1 -9284.328,E2 -9284.328} C_VEL
LIN {X 0,Y 433.712,Z 318.694,A -85,B 0,C 180,E1 -9285.747,E2 -9285.747} C_VEL
LIN {X 0,Y 434.414,Z 309.274,A -85,B 0,C 180,E1 -9286.929,E2 -9286.929} C_VEL
LIN {X 0,Y 435,Z 298.774,A -85,B 0,C 180,E1 -9287.997,E2 -9287.997} C_VEL
LIN {X 0,Y 435.756,Z 287.047,A -85,B 0,C 180,E1 -9288.939,E2 -9288.939} C_VEL
LIN {X 0,Y 436.167,Z 275.575,A -85,B 0,C 180,E1 -9289.654,E2 -9289.654} C_VEL
LIN {X 0,Y 436.283,Z 269.055,A -85,B 0,C 180,E1 -9289.982,E2 -9289.982} C_VEL
LIN {X 0,Y 433.381,Z 257.284,A -85,B 0,C 180,E1 -9290.577,E2 -9290.577} C_VEL
LIN {X 0,Y 431.524,Z 250.503,A -85,B 0,C 180,E1 -9290.879,E2 -9290.879} C_VEL
LIN {X 0,Y 431.651,Z 246.889,A -85,B 0,C 180,E1 -9294.247,E2 -9294.247} C_VEL
LIN {X 0,Y 431.697,Z 243.92,A -85,B 0,C 180,E1 -9297.117,E2 -9297.117} C_VEL
LIN {X 0,Y 431.777,Z 240.656,A -85,B 0,C 180,E1 -9300.381,E2 -9300.381} C_VEL
LIN {X 0,Y 431.868,Z 237.225,A -85,B 0,C 180,E1 -9303.906,E2 -9303.906} C_VEL
LIN {X 0,Y 431.937,Z 235.374,A -85,B 0,C 180,E1 -9305.854,E2 -9305.854} C_VEL
LIN {X 0,Y 432.032,Z 234.673,A -85,B 0,C 180,E1 -9307.145,E2 -9307.145} C_VEL
LIN {X 0,Y 432.239,Z 234.645,A -85,B 0,C 180,E1 -9309.353,E2 -9309.353} C_VEL
LIN {X 0,Y 432.321,Z 234.632,A -85,B 0,C 180,E1 -9311.796,E2 -9311.796} C_VEL
LIN {X 0,Y 432.327,Z 234.635,A -85,B 0,C 180,E1 -9314.346,E2 -9314.346} C_VEL
LIN {X 0,Y 432.309,Z 234.634,A -85,B 0,C 180,E1 -9317.015,E2 -9317.015} C_VEL
LIN {X 0,Y 432.324,Z 234.633,A -85,B 0,C 180,E1 -9319.82,E2 -9319.82} C_VEL
LIN {X 0,Y 432.307,Z 234.633,A -85,B 0,C 180,E1 -9323.022,E2 -9323.022} C_VEL
LIN {X 0,Y 432.351,Z 234.63,A -85,B 0,C 180,E1 -9325.995,E2 -9325.995} C_VEL
LIN {X 0,Y 432.338,Z 234.631,A -85,B 0,C 180,E1 -9329.489,E2 -9329.489} C_VEL
LIN {X 0,Y 432.383,Z 234.624,A -85,B 0,C 180,E1 -9332.927,E2 -9332.927} C_VEL
LIN {X 0,Y 432.361,Z 234.63,A -85,B 0,C 180,E1 -9336.023,E2 -9336.023} C_VEL
LIN {X 0,Y 432.339,Z 234.634,A -85,B 0,C 180,E1 -9339.045,E2 -9339.045} C_VEL
LIN {X 0,Y 432.366,Z 234.627,A -85,B 0,C 180,E1 -9342.01,E2 -9342.01} C_VEL
LIN {X 0,Y 432.384,Z 234.624,A -85,B 0,C 180,E1 -9344.926,E2 -9344.926} C_VEL
LIN {X 0,Y 432.447,Z 234.617,A -85,B 0,C 180,E1 -9347.803,E2 -9347.803} C_VEL
LIN {X 0,Y 432.48,Z 234.612,A -85,B 0,C 180,E1 -9351.59,E2 -9351.59} C_VEL
LIN {X 0,Y 432.594,Z 234.599,A -85,B 0,C 180,E1 -9354.406,E2 -9354.406} C_VEL
LIN {X 0,Y 432.595,Z 234.597,A -85,B 0,C 180,E1 -9358.138,E2 -9358.138} C_VEL
LIN {X 0,Y 432.718,Z 234.584,A -85,B 0,C 180,E1 -9360,E2 -9360} C_VEL
LIN {X 0,Y 432.595,Z 234.598,A -85,B 0,C 180,E1 -9362.794,E2 -9362.794} C_VEL
LIN {X 0,Y 432.565,Z 234.602,A -85,B 0,C 180,E1 -9366.53,E2 -9366.53} C_VEL
LIN {X 0,Y 432.43,Z 234.618,A -85,B 0,C 180,E1 -9369.353,E2 -9369.353} C_VEL
LIN {X 0,Y 432.419,Z 234.618,A -85,B 0,C 180,E1 -9372.804,E2 -9372.804} C_VEL
LIN {X 0,Y 432.401,Z 234.62,A -85,B 0,C 180,E1 -9376.479,E2 -9376.479} C_VEL
LIN {X 0,Y 432.327,Z 234.631,A -85,B 0,C 180,E1 -9379.961,E2 -9379.961} C_VEL
LIN {X 0,Y 432.307,Z 234.634,A -85,B 0,C 180,E1 -9382.965,E2 -9382.965} C_VEL
LIN {X 0,Y 432.354,Z 234.628,A -85,B 0,C 180,E1 -9386.033,E2 -9386.033} C_VEL
LIN {X 0,Y 432.342,Z 234.63,A -85,B 0,C 180,E1 -9389.188,E2 -9389.188} C_VEL
LIN {X 0,Y 432.321,Z 234.633,A -85,B 0,C 180,E1 -9392.295,E2 -9392.295} C_VEL
LIN {X 0,Y 432.33,Z 234.633,A -85,B 0,C 180,E1 -9394.678,E2 -9394.678} C_VEL
LIN {X 0,Y 432.328,Z 234.633,A -85,B 0,C 180,E1 -9398.151,E2 -9398.151} C_VEL
LIN {X 0,Y 432.316,Z 234.636,A -85,B 0,C 180,E1 -9401.602,E2 -9401.602} C_VEL
LIN {X 0,Y 432.325,Z 234.634,A -85,B 0,C 180,E1 -9404.349,E2 -9404.349} C_VEL
LIN {X 0,Y 432.351,Z 234.72,A -85,B 0,C 180,E1 -9407.422,E2 -9407.422} C_VEL
LIN {X 0,Y 433.395,Z 240.141,A -85,B 0,C 180,E1 -9410.244,E2 -9410.244} C_VEL
LIN {X 0,Y 434.383,Z 246.305,A -85,B 0,C 180,E1 -9413.23,E2 -9413.23} C_VEL
LIN {X 0,Y 434.38,Z 250.141,A -85,B 0,C 180,E1 -9414.947,E2 -9414.947} C_VEL
LIN {X 0,Y 433.923,Z 256.6,A -85,B 0,C 180,E1 -9417.693,E2 -9417.693} C_VEL
LIN {X 0,Y 433.358,Z 264.446,A -85,B 0,C 180,E1 -9420.889,E2 -9420.889} C_VEL
LIN {X 0,Y 433.039,Z 271.294,A -85,B 0,C 180,E1 -9423.6,E2 -9423.6} C_VEL
LIN {X 0,Y 432.529,Z 280.268,A -85,B 0,C 180,E1 -9427.049,E2 -9427.049} C_VEL
LIN {X 0,Y 432.208,Z 288.211,A -85,B 0,C 180,E1 -9430.035,E2 -9430.035} C_VEL
LIN {X 0,Y 431.849,Z 297.108,A -85,B 0,C 180,E1 -9433.297,E2 -9433.297} C_VEL
LIN {X 0,Y 433.988,Z 310.525,A -85,B 0,C 180,E1 -9433.751,E2 -9433.751} C_VEL
LIN {X 0,Y 435.568,Z 321.341,A -85,B 0,C 180,E1 -9434.261,E2 -9434.261} C_VEL
LIN {X 0,Y 435.079,Z 333.019,A -85,B 0,C 180,E1 -9434.903,E2 -9434.903} C_VEL
LIN {X 0,Y 434.389,Z 344.413,A -85,B 0,C 180,E1 -9435.717,E2 -9435.717} C_VEL
LIN {X 0,Y 433.729,Z 355.687,A -85,B 0,C 180,E1 -9436.738,E2 -9436.738} C_VEL
LIN {X 0,Y 433.216,Z 365.364,A -85,B 0,C 180,E1 -9437.827,E2 -9437.827} C_VEL
LIN {X 0,Y 432.586,Z 373.89,A -85,B 0,C 180,E1 -9438.996,E2 -9438.996} C_VEL
LIN {X 0,Y 432.1,Z 382.221,A -85,B 0,C 180,E1 -9440.405,E2 -9440.405} C_VEL
LIN {X 0,Y 431.709,Z 388.941,A -85,B 0,C 180,E1 -9441.812,E2 -9441.812} C_VEL
LIN {X 0,Y 431.446,Z 395.098,A -85,B 0,C 180,E1 -9443.454,E2 -9443.454} C_VEL
LIN {X 0,Y 431.368,Z 399.105,A -85,B 0,C 180,E1 -9444.86,E2 -9444.86} C_VEL
LIN {X 0,Y 431.21,Z 402.059,A -85,B 0,C 180,E1 -9446.263,E2 -9446.263} C_VEL
LIN {X 0,Y 431.279,Z 403.474,A -85,B 0,C 180,E1 -9447.199,E2 -9447.199} C_VEL
LIN {X 0,Y 431.197,Z 405.092,A -85,B 0,C 180,E1 -9449.067,E2 -9449.067} C_VEL
LIN {X 0,Y 431.216,Z 405.312,A -85,B 0,C 180,E1 -9450.001,E2 -9450.001} C_VEL
LIN {X 0,Y 431.198,Z 405.093,A -85,B 0,C 180,E1 -9450.935,E2 -9450.935} C_VEL
LIN {X 0,Y 431.28,Z 403.481,A -85,B 0,C 180,E1 -9452.803,E2 -9452.803} C_VEL
LIN {X 0,Y 431.21,Z 402.067,A -85,B 0,C 180,E1 -9453.739,E2 -9453.739} C_VEL
LIN {X 0,Y 431.369,Z 399.112,A -85,B 0,C 180,E1 -9455.142,E2 -9455.142} C_VEL
LIN {X 0,Y 431.442,Z 395.103,A -85,B 0,C 180,E1 -9456.549,E2 -9456.549} C_VEL
LIN {X 0,Y 431.713,Z 388.948,A -85,B 0,C 180,E1 -9458.191,E2 -9458.191} C_VEL
LIN {X 0,Y 432.104,Z 382.23,A -85,B 0,C 180,E1 -9459.598,E2 -9459.598} C_VEL
LIN {X 0,Y 432.589,Z 373.898,A -85,B 0,C 180,E1 -9461.006,E2 -9461.006} C_VEL
LIN {X 0,Y 433.201,Z 365.37,A -85,B 0,C 180,E1 -9462.177,E2 -9462.177} C_VEL
LIN {X 0,Y 433.812,Z 355.382,A -85,B 0,C 180,E1 -9463.294,E2 -9463.294} C_VEL
LIN {X 0,Y 434.445,Z 344.42,A -85,B 0,C 180,E1 -9464.284,E2 -9464.284} C_VEL
LIN {X 0,Y 435.067,Z 333.01,A -85,B 0,C 180,E1 -9465.1,E2 -9465.1} C_VEL
LIN {X 0,Y 435.598,Z 321.308,A -85,B 0,C 180,E1 -9465.74,E2 -9465.74} C_VEL
LIN {X 0,Y 433.573,Z 307.751,A -85,B 0,C 180,E1 -9466.357,E2 -9466.357} C_VEL
LIN {X 0,Y 431.841,Z 297,A -85,B 0,C 180,E1 -9466.722,E2 -9466.722} C_VEL
LIN {X 0,Y 432.215,Z 288.252,A -85,B 0,C 180,E1 -9469.968,E2 -9469.968} C_VEL
LIN {X 0,Y 432.521,Z 280.265,A -85,B 0,C 180,E1 -9472.954,E2 -9472.954} C_VEL
LIN {X 0,Y 433.018,Z 271.202,A -85,B 0,C 180,E1 -9476.396,E2 -9476.396} C_VEL
LIN {X 0,Y 433.35,Z 264.186,A -85,B 0,C 180,E1 -9479.114,E2 -9479.114} C_VEL
LIN {X 0,Y 433.876,Z 256.188,A -85,B 0,C 180,E1 -9482.314,E2 -9482.314} C_VEL
LIN {X 0,Y 434.326,Z 249.56,A -85,B 0,C 180,E1 -9485.062,E2 -9485.062} C_VEL
LIN {X 0,Y 434.26,Z 245.581,A -85,B 0,C 180,E1 -9486.786,E2 -9486.786} C_VEL
LIN {X 0,Y 433.194,Z 239.193,A -85,B 0,C 180,E1 -9489.755,E2 -9489.755} C_VEL
LIN {X 0,Y 432.375,Z 234.631,A -85,B 0,C 180,E1 -9492.107,E2 -9492.107} C_VEL
LIN {X 0,Y 432.34,Z 234.636,A -85,B 0,C 180,E1 -9495.665,E2 -9495.665} C_VEL
LIN {X 0,Y 432.339,Z 234.631,A -85,B 0,C 180,E1 -9498.399,E2 -9498.399} C_VEL
LIN {X 0,Y 432.341,Z 234.629,A -85,B 0,C 180,E1 -9501.85,E2 -9501.85} C_VEL
LIN {X 0,Y 432.333,Z 234.629,A -85,B 0,C 180,E1 -9505.322,E2 -9505.322} C_VEL
LIN {X 0,Y 432.323,Z 234.634,A -85,B 0,C 180,E1 -9508.654,E2 -9508.654} C_VEL
LIN {X 0,Y 432.354,Z 234.63,A -85,B 0,C 180,E1 -9511.875,E2 -9511.875} C_VEL
LIN {X 0,Y 432.386,Z 234.625,A -85,B 0,C 180,E1 -9515.539,E2 -9515.539} C_VEL
LIN {X 0,Y 432.357,Z 234.628,A -85,B 0,C 180,E1 -9519.046,E2 -9519.046} C_VEL
LIN {X 0,Y 432.356,Z 234.63,A -85,B 0,C 180,E1 -9522.01,E2 -9522.01} C_VEL
LIN {X 0,Y 432.354,Z 234.626,A -85,B 0,C 180,E1 -9524.925,E2 -9524.925} C_VEL
LIN {X 0,Y 432.461,Z 234.619,A -85,B 0,C 180,E1 -9527.804,E2 -9527.804} C_VEL
LIN {X 0,Y 432.468,Z 234.618,A -85,B 0,C 180,E1 -9531.59,E2 -9531.59} C_VEL
LIN {X 0,Y 432.599,Z 234.598,A -85,B 0,C 180,E1 -9534.406,E2 -9534.406} C_VEL
LIN {X 0,Y 432.61,Z 234.598,A -85,B 0,C 180,E1 -9538.138,E2 -9538.138} C_VEL
LIN {X 0,Y 432.736,Z 234.582,A -85,B 0,C 180,E1 -9540,E2 -9540} C_VEL
LIN {X 0,Y 432.586,Z 234.599,A -85,B 0,C 180,E1 -9542.794,E2 -9542.794} C_VEL
LIN {X 0,Y 432.514,Z 234.606,A -85,B 0,C 180,E1 -9546.531,E2 -9546.531} C_VEL
LIN {X 0,Y 432.437,Z 234.62,A -85,B 0,C 180,E1 -9549.353,E2 -9549.353} C_VEL
LIN {X 0,Y 432.439,Z 234.62,A -85,B 0,C 180,E1 -9552.803,E2 -9552.803} C_VEL
LIN {X 0,Y 432.42,Z 234.622,A -85,B 0,C 180,E1 -9556.478,E2 -9556.478} C_VEL
LIN {X 0,Y 432.346,Z 234.629,A -85,B 0,C 180,E1 -9559.96,E2 -9559.96} C_VEL
LIN {X 0,Y 432.317,Z 234.637,A -85,B 0,C 180,E1 -9562.965,E2 -9562.965} C_VEL
LIN {X 0,Y 432.312,Z 234.632,A -85,B 0,C 180,E1 -9566.036,E2 -9566.036} C_VEL
LIN {X 0,Y 432.33,Z 234.631,A -85,B 0,C 180,E1 -9569.189,E2 -9569.189} C_VEL
LIN {X 0,Y 432.33,Z 234.634,A -85,B 0,C 180,E1 -9572.443,E2 -9572.443} C_VEL
LIN {X 0,Y 432.35,Z 234.629,A -85,B 0,C 180,E1 -9575.631,E2 -9575.631} C_VEL
LIN {X 0,Y 432.34,Z 234.633,A -85,B 0,C 180,E1 -9578.713,E2 -9578.713} C_VEL
LIN {X 0,Y 432.331,Z 234.632,A -85,B 0,C 180,E1 -9581.798,E2 -9581.798} C_VEL
LIN {X 0,Y 432.339,Z 234.634,A -85,B 0,C 180,E1 -9584.347,E2 -9584.347} C_VEL
LIN {X 0,Y 432.308,Z 234.632,A -85,B 0,C 180,E1 -9587.018,E2 -9587.018} C_VEL
LIN {X 0,Y 432.294,Z 234.639,A -85,B 0,C 180,E1 -9589.828,E2 -9589.828} C_VEL
LIN {X 0,Y 432.311,Z 234.633,A -85,B 0,C 180,E1 -9593.021,E2 -9593.021} C_VEL
LIN {X 0,Y 432.339,Z 234.632,A -85,B 0,C 180,E1 -9596.001,E2 -9596.001} C_VEL
LIN {X 0,Y 432.205,Z 234.647,A -85,B 0,C 180,E1 -9598.643,E2 -9598.643} C_VEL
LIN {X 0,Y 431.903,Z 234.689,A -85,B 0,C 180,E1 -9601.841,E2 -9601.841} C_VEL
LIN {X 0,Y 431.77,Z 235.104,A -85,B 0,C 180,E1 -9602.885,E2 -9602.885} C_VEL
LIN {X 0,Y 431.759,Z 238.166,A -85,B 0,C 180,E1 -9605.986,E2 -9605.986} C_VEL
LIN {X 0,Y 431.623,Z 241.236,A -85,B 0,C 180,E1 -9609.008,E2 -9609.008} C_VEL
LIN {X 0,Y 431.592,Z 244.309,A -85,B 0,C 180,E1 -9611.976,E2 -9611.976} C_VEL
LIN {X 0,Y 431.604,Z 247.418,A -85,B 0,C 180,E1 -9614.897,E2 -9614.897} C_VEL
LIN {X 0,Y 431.614,Z 250.383,A -85,B 0,C 180,E1 -9617.548,E2 -9617.548} C_VEL
LIN {X 0,Y 435.005,Z 264.831,A -85,B 0,C 180,E1 -9618.156,E2 -9618.156} C_VEL
LIN {X 0,Y 435.909,Z 270.247,A -85,B 0,C 180,E1 -9618.431,E2 -9618.431} C_VEL
LIN {X 0,Y 435.479,Z 281.921,A -85,B 0,C 180,E1 -9619.068,E2 -9619.068} C_VEL
LIN {X 0,Y 434.897,Z 293.236,A -85,B 0,C 180,E1 -9619.877,E2 -9619.877} C_VEL
LIN {X 0,Y 434.224,Z 304.922,A -85,B 0,C 180,E1 -9620.942,E2 -9620.942} C_VEL
LIN {X 0,Y 433.732,Z 314.831,A -85,B 0,C 180,E1 -9622.082,E2 -9622.082} C_VEL
LIN {X 0,Y 433.051,Z 324.549,A -85,B 0,C 180,E1 -9623.476,E2 -9623.476} C_VEL
LIN {X 0,Y 432.492,Z 332.367,A -85,B 0,C 180,E1 -9624.871,E2 -9624.871} C_VEL
LIN {X 0,Y 431.996,Z 338.618,A -85,B 0,C 180,E1 -9626.268,E2 -9626.268} C_VEL
LIN {X 0,Y 431.713,Z 342.032,A -85,B 0,C 180,E1 -9627.194,E2 -9627.194} C_VEL
LIN {X 0,Y 430.868,Z 344.442,A -85,B 0,C 180,E1 -9627.903,E2 -9627.903} C_VEL
LIN {X 0,Y 427.859,Z 347.88,A -85,B 0,C 180,E1 -9629.078,E2 -9629.078} C_VEL
LIN {X 0,Y 425.408,Z 350.056,A -85,B 0,C 180,E1 -9630.051,E2 -9630.051} C_VEL
LIN {X 0,Y 424.361,Z 351.322,A -85,B 0,C 180,E1 -9630.818,E2 -9630.818} C_VEL
LIN {X 0,Y 424.274,Z 351.665,A -85,B 0,C 180,E1 -9631.081,E2 -9631.081} C_VEL
LIN {X 0,Y 424.299,Z 352.658,A -85,B 0,C 180,E1 -9631.897,E2 -9631.897} C_VEL
LIN {X 0,Y 424.335,Z 353.382,A -85,B 0,C 180,E1 -9632.847,E2 -9632.847} C_VEL
LIN {X 0,Y 424.316,Z 353.73,A -85,B 0,C 180,E1 -9633.797,E2 -9633.797} C_VEL
LIN {X 0,Y 424.336,Z 353.288,A -85,B 0,C 180,E1 -9635.702,E2 -9635.702} C_VEL
LIN {X 0,Y 424.381,Z 352.443,A -85,B 0,C 180,E1 -9636.655,E2 -9636.655} C_VEL
LIN {X 0,Y 424.517,Z 349.568,A -85,B 0,C 180,E1 -9638.567,E2 -9638.567} C_VEL
LIN {X 0,Y 424.703,Z 346.263,A -85,B 0,C 180,E1 -9640.005,E2 -9640.005} C_VEL
LIN {X 0,Y 425.034,Z 341.877,A -85,B 0,C 180,E1 -9641.443,E2 -9641.443} C_VEL
LIN {X 0,Y 425.436,Z 336.109,A -85,B 0,C 180,E1 -9642.926,E2 -9642.926} C_VEL
LIN {X 0,Y 425.992,Z 329.245,A -85,B 0,C 180,E1 -9644.326,E2 -9644.326} C_VEL
LIN {X 0,Y 426.703,Z 320.427,A -85,B 0,C 180,E1 -9645.768,E2 -9645.768} C_VEL
LIN {X 0,Y 427.416,Z 311.356,A -85,B 0,C 180,E1 -9646.968,E2 -9646.968} C_VEL
LIN {X 0,Y 428.012,Z 301.363,A -85,B 0,C 180,E1 -9648.046,E2 -9648.046} C_VEL
LIN {X 0,Y 428.795,Z 290.034,A -85,B 0,C 180,E1 -9649.01,E2 -9649.01} C_VEL
LIN {X 0,Y 429.295,Z 277.917,A -85,B 0,C 180,E1 -9649.822,E2 -9649.822} C_VEL
LIN {X 0,Y 429.494,Z 270.343,A -85,B 0,C 180,E1 -9650.222,E2 -9650.222} C_VEL
LIN {X 0,Y 426.541,Z 258.306,A -85,B 0,C 180,E1 -9650.852,E2 -9650.852} C_VEL
LIN {X 0,Y 424.451,Z 250.949,A -85,B 0,C 180,E1 -9651.167,E2 -9651.167} C_VEL
LIN {X 0,Y 424.596,Z 247.46,A -85,B 0,C 180,E1 -9654.442,E2 -9654.442} C_VEL
LIN {X 0,Y 424.657,Z 244.225,A -85,B 0,C 180,E1 -9657.605,E2 -9657.605} C_VEL
LIN {X 0,Y 424.725,Z 241.013,A -85,B 0,C 180,E1 -9660.86,E2 -9660.86} C_VEL
LIN {X 0,Y 424.844,Z 237.767,A -85,B 0,C 180,E1 -9664.223,E2 -9664.223} C_VEL
LIN {X 0,Y 424.905,Z 235.602,A -85,B 0,C 180,E1 -9666.542,E2 -9666.542} C_VEL
LIN {X 0,Y 425.179,Z 235.525,A -85,B 0,C 180,E1 -9669.023,E2 -9669.023} C_VEL
LIN {X 0,Y 425.279,Z 235.509,A -85,B 0,C 180,E1 -9671.956,E2 -9671.956} C_VEL
LIN {X 0,Y 425.278,Z 235.51,A -85,B 0,C 180,E1 -9675.282,E2 -9675.282} C_VEL
LIN {X 0,Y 425.259,Z 235.512,A -85,B 0,C 180,E1 -9678.619,E2 -9678.619} C_VEL
LIN {X 0,Y 425.293,Z 235.51,A -85,B 0,C 180,E1 -9681.1,E2 -9681.1} C_VEL
LIN {X 0,Y 425.292,Z 235.509,A -85,B 0,C 180,E1 -9684.663,E2 -9684.663} C_VEL
LIN {X 0,Y 425.255,Z 235.512,A -85,B 0,C 180,E1 -9688.072,E2 -9688.072} C_VEL
LIN {X 0,Y 425.322,Z 235.504,A -85,B 0,C 180,E1 -9691.367,E2 -9691.367} C_VEL
LIN {X 0,Y 425.286,Z 235.509,A -85,B 0,C 180,E1 -9694.554,E2 -9694.554} C_VEL
LIN {X 0,Y 425.277,Z 235.512,A -85,B 0,C 180,E1 -9697.66,E2 -9697.66} C_VEL
LIN {X 0,Y 425.351,Z 235.505,A -85,B 0,C 180,E1 -9700.703,E2 -9700.703} C_VEL
LIN {X 0,Y 425.377,Z 235.499,A -85,B 0,C 180,E1 -9703.688,E2 -9703.688} C_VEL
LIN {X 0,Y 425.4,Z 235.496,A -85,B 0,C 180,E1 -9707.598,E2 -9707.598} C_VEL
LIN {X 0,Y 425.43,Z 235.49,A -85,B 0,C 180,E1 -9711.45,E2 -9711.45} C_VEL
LIN {X 0,Y 425.569,Z 235.475,A -85,B 0,C 180,E1 -9714.313,E2 -9714.313} C_VEL
LIN {X 0,Y 425.565,Z 235.473,A -85,B 0,C 180,E1 -9718.107,E2 -9718.107} C_VEL
LIN {X 0,Y 425.687,Z 235.459,A -85,B 0,C 180,E1 -9720,E2 -9720} C_VEL
LIN {X 0,Y 425.546,Z 235.476,A -85,B 0,C 180,E1 -9722.84,E2 -9722.84} C_VEL
LIN {X 0,Y 425.568,Z 235.475,A -85,B 0,C 180,E1 -9725.686,E2 -9725.686} C_VEL
LIN {X 0,Y 425.43,Z 235.494,A -85,B 0,C 180,E1 -9728.55,E2 -9728.55} C_VEL
LIN {X 0,Y 425.4,Z 235.494,A -85,B 0,C 180,E1 -9732.402,E2 -9732.402} C_VEL
LIN {X 0,Y 425.377,Z 235.495,A -85,B 0,C 180,E1 -9736.312,E2 -9736.312} C_VEL
LIN {X 0,Y 425.317,Z 235.503,A -85,B 0,C 180,E1 -9739.636,E2 -9739.636} C_VEL
LIN {X 0,Y 425.295,Z 235.51,A -85,B 0,C 180,E1 -9743.366,E2 -9743.366} C_VEL
LIN {X 0,Y 425.338,Z 235.506,A -85,B 0,C 180,E1 -9746.845,E2 -9746.845} C_VEL
LIN {X 0,Y 425.308,Z 235.507,A -85,B 0,C 180,E1 -9749.718,E2 -9749.718} C_VEL
LIN {X 0,Y 425.274,Z 235.512,A -85,B 0,C 180,E1 -9753.049,E2 -9753.049} C_VEL
LIN {X 0,Y 425.273,Z 235.51,A -85,B 0,C 180,E1 -9755.93,E2 -9755.93} C_VEL
LIN {X 0,Y 425.284,Z 235.509,A -85,B 0,C 180,E1 -9759.044,E2 -9759.044} C_VEL
LIN {X 0,Y 425.262,Z 235.512,A -85,B 0,C 180,E1 -9762.655,E2 -9762.655} C_VEL
LIN {X 0,Y 425.254,Z 235.517,A -85,B 0,C 180,E1 -9766.045,E2 -9766.045} C_VEL
LIN {X 0,Y 425.3,Z 235.541,A -85,B 0,C 180,E1 -9767.005,E2 -9767.005} C_VEL
LIN {X 0,Y 426.372,Z 241.163,A -85,B 0,C 180,E1 -9769.998,E2 -9769.998} C_VEL
LIN {X 0,Y 427.393,Z 247.462,A -85,B 0,C 180,E1 -9773.118,E2 -9773.118} C_VEL
LIN {X 0,Y 427.353,Z 252.29,A -85,B 0,C 180,E1 -9775.313,E2 -9775.313} C_VEL
LIN {X 0,Y 426.834,Z 259.027,A -85,B 0,C 180,E1 -9778.206,E2 -9778.206} C_VEL
LIN {X 0,Y 426.237,Z 268.163,A -85,B 0,C 180,E1 -9781.973,E2 -9781.973} C_VEL
LIN {X 0,Y 425.696,Z 276.368,A -85,B 0,C 180,E1 -9785.233,E2 -9785.233} C_VEL
LIN {X 0,Y 425.274,Z 285.248,A -85,B 0,C 180,E1 -9788.682,E2 -9788.682} C_VEL
LIN {X 0,Y 424.927,Z 293.144,A -85,B 0,C 180,E1 -9791.686,E2 -9791.686} C_VEL
LIN {X 0,Y 424.775,Z 296.617,A -85,B 0,C 180,E1 -9792.994,E2 -9792.994} C_VEL
LIN {X 0,Y 427.043,Z 311.053,A -85,B 0,C 180,E1 -9793.515,E2 -9793.515} C_VEL
LIN {X 0,Y 428.676,Z 322.118,A -85,B 0,C 180,E1 -9794.063,E2 -9794.063} C_VEL
LIN {X 0,Y 428.073,Z 334.357,A -85,B 0,C 180,E1 -9794.772,E2 -9794.772} C_VEL
LIN {X 0,Y 427.385,Z 345.412,A -85,B 0,C 180,E1 -9795.6,E2 -9795.6} C_VEL
LIN {X 0,Y 426.693,Z 356.717,A -85,B 0,C 180,E1 -9796.67,E2 -9796.67} C_VEL
LIN {X 0,Y 426.099,Z 366.738,A -85,B 0,C 180,E1 -9797.862,E2 -9797.862} C_VEL
LIN {X 0,Y 425.389,Z 376.455,A -85,B 0,C 180,E1 -9799.29,E2 -9799.29} C_VEL
LIN {X 0,Y 424.9,Z 384.202,A -85,B 0,C 180,E1 -9800.721,E2 -9800.721} C_VEL
LIN {X 0,Y 424.463,Z 391.347,A -85,B 0,C 180,E1 -9802.39,E2 -9802.39} C_VEL
LIN {X 0,Y 424.276,Z 396.488,A -85,B 0,C 180,E1 -9803.946,E2 -9803.946} C_VEL
LIN {X 0,Y 424.226,Z 399.754,A -85,B 0,C 180,E1 -9805.25,E2 -9805.25} C_VEL
LIN {X 0,Y 424.12,Z 401.63,A -85,B 0,C 180,E1 -9806.201,E2 -9806.201} C_VEL
LIN {X 0,Y 424.191,Z 403.046,A -85,B 0,C 180,E1 -9807.152,E2 -9807.152} C_VEL
LIN {X 0,Y 424.115,Z 404.665,A -85,B 0,C 180,E1 -9809.052,E2 -9809.052} C_VEL
LIN {X 0,Y 424.13,Z 404.885,A -85,B 0,C 180,E1 -9810.001,E2 -9810.001} C_VEL
LIN {X 0,Y 424.115,Z 404.667,A -85,B 0,C 180,E1 -9810.951,E2 -9810.951} C_VEL
LIN {X 0,Y 424.192,Z 403.054,A -85,B 0,C 180,E1 -9812.85,E2 -9812.85} C_VEL
LIN {X 0,Y 424.12,Z 401.64,A -85,B 0,C 180,E1 -9813.802,E2 -9813.802} C_VEL
LIN {X 0,Y 424.28,Z 398.684,A -85,B 0,C 180,E1 -9815.229,E2 -9815.229} C_VEL
LIN {X 0,Y 424.36,Z 394.675,A -85,B 0,C 180,E1 -9816.659,E2 -9816.659} C_VEL
LIN {X 0,Y 424.652,Z 388.52,A -85,B 0,C 180,E1 -9818.328,E2 -9818.328} C_VEL
LIN {X 0,Y 425.048,Z 381.801,A -85,B 0,C 180,E1 -9819.759,E2 -9819.759} C_VEL
LIN {X 0,Y 425.584,Z 373.471,A -85,B 0,C 180,E1 -9821.19,E2 -9821.19} C_VEL
LIN {X 0,Y 426.216,Z 364.942,A -85,B 0,C 180,E1 -9822.379,E2 -9822.379} C_VEL
LIN {X 0,Y 426.833,Z 355.478,A -85,B 0,C 180,E1 -9823.461,E2 -9823.461} C_VEL
LIN {X 0,Y 427.42,Z 345.424,A -85,B 0,C 180,E1 -9824.402,E2 -9824.402} C_VEL
LIN {X 0,Y 428.089,Z 334.358,A -85,B 0,C 180,E1 -9825.23,E2 -9825.23} C_VEL
LIN {X 0,Y 428.678,Z 322.099,A -85,B 0,C 180,E1 -9825.94,E2 -9825.94} C_VEL
LIN {X 0,Y 426.812,Z 309.318,A -85,B 0,C 180,E1 -9826.557,E2 -9826.557} C_VEL
LIN {X 0,Y 424.782,Z 296.645,A -85,B 0,C 180,E1 -9827.008,E2 -9827.008} C_VEL
LIN {X 0,Y 425.13,Z 289.041,A -85,B 0,C 180,E1 -9829.877,E2 -9829.877} C_VEL
LIN {X 0,Y 425.434,Z 281.245,A -85,B 0,C 180,E1 -9832.845,E2 -9832.845} C_VEL
LIN {X 0,Y 425.973,Z 271.907,A -85,B 0,C 180,E1 -9836.454,E2 -9836.454} C_VEL
LIN {X 0,Y 426.317,Z 265.188,A -85,B 0,C 180,E1 -9839.105,E2 -9839.105} C_VEL
LIN {X 0,Y 426.863,Z 257.215,A -85,B 0,C 180,E1 -9842.351,E2 -9842.351} C_VEL
LIN {X 0,Y 427.355,Z 250.608,A -85,B 0,C 180,E1 -9845.142,E2 -9845.142} C_VEL
LIN {X 0,Y 427.253,Z 246.639,A -85,B 0,C 180,E1 -9846.899,E2 -9846.899} C_VEL
LIN {X 0,Y 426.146,Z 240.044,A -85,B 0,C 180,E1 -9850.031,E2 -9850.031} C_VEL
LIN {X 0,Y 425.345,Z 235.506,A -85,B 0,C 180,E1 -9852.359,E2 -9852.359} C_VEL
LIN {X 0,Y 425.268,Z 235.517,A -85,B 0,C 180,E1 -9856.045,E2 -9856.045} C_VEL
LIN {X 0,Y 425.281,Z 235.511,A -85,B 0,C 180,E1 -9858.622,E2 -9858.622} C_VEL
LIN {X 0,Y 425.304,Z 235.508,A -85,B 0,C 180,E1 -9861.102,E2 -9861.102} C_VEL
LIN {X 0,Y 425.3,Z 235.511,A -85,B 0,C 180,E1 -9864.664,E2 -9864.664} C_VEL
LIN {X 0,Y 425.268,Z 235.512,A -85,B 0,C 180,E1 -9868.073,E2 -9868.073} C_VEL
LIN {X 0,Y 425.32,Z 235.504,A -85,B 0,C 180,E1 -9871.367,E2 -9871.367} C_VEL
LIN {X 0,Y 425.28,Z 235.511,A -85,B 0,C 180,E1 -9874.554,E2 -9874.554} C_VEL
LIN {X 0,Y 425.312,Z 235.508,A -85,B 0,C 180,E1 -9876.635,E2 -9876.635} C_VEL
LIN {X 0,Y 425.336,Z 235.506,A -85,B 0,C 180,E1 -9880.365,E2 -9880.365} C_VEL
LIN {X 0,Y 425.33,Z 235.504,A -85,B 0,C 180,E1 -9883.686,E2 -9883.686} C_VEL
LIN {X 0,Y 425.4,Z 235.492,A -85,B 0,C 180,E1 -9887.098,E2 -9887.098} C_VEL
LIN {X 0,Y 425.392,Z 235.495,A -85,B 0,C 180,E1 -9890.49,E2 -9890.49} C_VEL
LIN {X 0,Y 425.518,Z 235.482,A -85,B 0,C 180,E1 -9893.361,E2 -9893.361} C_VEL
LIN {X 0,Y 425.371,Z 235.5,A -85,B 0,C 180,E1 -9895.261,E2 -9895.261} C_VEL
LIN {X 0,Y 425.58,Z 235.473,A -85,B 0,C 180,E1 -9898.107,E2 -9898.107} C_VEL
LIN {X 0,Y 425.705,Z 235.458,A -85,B 0,C 180,E1 -9900,E2 -9900} C_VEL
LIN {X 0,Y 425.54,Z 235.477,A -85,B 0,C 180,E1 -9902.84,E2 -9902.84} C_VEL
LIN {X 0,Y 425.476,Z 235.483,A -85,B 0,C 180,E1 -9906.64,E2 -9906.64} C_VEL
LIN {X 0,Y 425.397,Z 235.496,A -85,B 0,C 180,E1 -9909.51,E2 -9909.51} C_VEL
LIN {X 0,Y 425.402,Z 235.498,A -85,B 0,C 180,E1 -9912.903,E2 -9912.903} C_VEL
LIN {X 0,Y 425.369,Z 235.501,A -85,B 0,C 180,E1 -9916.604,E2 -9916.604} C_VEL
LIN {X 0,Y 425.336,Z 235.503,A -85,B 0,C 180,E1 -9919.635,E2 -9919.635} C_VEL
LIN {X 0,Y 425.295,Z 235.508,A -85,B 0,C 180,E1 -9922.339,E2 -9922.339} C_VEL
LIN {X 0,Y 425.258,Z 235.511,A -85,B 0,C 180,E1 -9925.448,E2 -9925.448} C_VEL
LIN {X 0,Y 425.308,Z 235.508,A -85,B 0,C 180,E1 -9928.858,E2 -9928.858} C_VEL
LIN {X 0,Y 425.271,Z 235.51,A -85,B 0,C 180,E1 -9931.927,E2 -9931.927} C_VEL
LIN {X 0,Y 425.305,Z 235.506,A -85,B 0,C 180,E1 -9935.336,E2 -9935.336} C_VEL
LIN {X 0,Y 425.299,Z 235.508,A -85,B 0,C 180,E1 -9938.899,E2 -9938.899} C_VEL
LIN {X 0,Y 425.29,Z 235.509,A -85,B 0,C 180,E1 -9941.956,E2 -9941.956} C_VEL
LIN {X 0,Y 425.29,Z 235.507,A -85,B 0,C 180,E1 -9945.283,E2 -9945.283} C_VEL
LIN {X 0,Y 425.252,Z 235.512,A -85,B 0,C 180,E1 -9948.617,E2 -9948.617} C_VEL
LIN {X 0,Y 425.285,Z 235.508,A -85,B 0,C 180,E1 -9951.098,E2 -9951.098} C_VEL
LIN {X 0,Y 425.302,Z 235.507,A -85,B 0,C 180,E1 -9954.663,E2 -9954.663} C_VEL
LIN {X 0,Y 425.187,Z 235.523,A -85,B 0,C 180,E1 -9958.065,E2 -9958.065} C_VEL
LIN {X 0,Y 424.904,Z 235.56,A -85,B 0,C 180,E1 -9961.335,E2 -9961.335} C_VEL
LIN {X 0,Y 424.762,Z 235.579,A -85,B 0,C 180,E1 -9962.4,E2 -9962.4} C_VEL
LIN {X 0,Y 424.703,Z 238.542,A -85,B 0,C 180,E1 -9965.561,E2 -9965.561} C_VEL
LIN {X 0,Y 424.59,Z 241.599,A -85,B 0,C 180,E1 -9968.643,E2 -9968.643} C_VEL
LIN {X 0,Y 424.53,Z 244.71,A -85,B 0,C 180,E1 -9971.666,E2 -9971.666} C_VEL
LIN {X 0,Y 424.546,Z 247.849,A -85,B 0,C 180,E1 -9974.64,E2 -9974.64} C_VEL
LIN {X 0,Y 424.58,Z 250.948,A -85,B 0,C 180,E1 -9977.3,E2 -9977.3} C_VEL
LIN {X 0,Y 427.772,Z 264.244,A -85,B 0,C 180,E1 -9977.861,E2 -9977.861} C_VEL
LIN {X 0,Y 429.036,Z 271.134,A -85,B 0,C 180,E1 -9978.217,E2 -9978.217} C_VEL
LIN {X 0,Y 428.58,Z 283.043,A -85,B 0,C 180,E1 -9978.889,E2 -9978.889} C_VEL
LIN {X 0,Y 427.971,Z 294.219,A -85,B 0,C 180,E1 -9979.711,E2 -9979.711} C_VEL
LIN {X 0,Y 427.285,Z 305.805,A -85,B 0,C 180,E1 -9980.794,E2 -9980.794} C_VEL
LIN {X 0,Y 426.748,Z 315.606,A -85,B 0,C 180,E1 -9981.952,E2 -9981.952} C_VEL
LIN {X 0,Y 426.049,Z 325.266,A -85,B 0,C 180,E1 -9983.368,E2 -9983.368} C_VEL
LIN {X 0,Y 425.479,Z 333.022,A -85,B 0,C 180,E1 -9984.786,E2 -9984.786} C_VEL
LIN {X 0,Y 424.963,Z 339.221,A -85,B 0,C 180,E1 -9986.206,E2 -9986.206} C_VEL
LIN {X 0,Y 424.627,Z 344.152,A -85,B 0,C 180,E1 -9987.627,E2 -9987.627} C_VEL
LIN {X 0,Y 424.348,Z 347.979,A -85,B 0,C 180,E1 -9989.05,E2 -9989.05} C_VEL
LIN {X 0,Y 424.282,Z 349.945,A -85,B 0,C 180,E1 -9989.999,E2 -9989.999} C_VEL
LIN {X 0,Y 424.274,Z 351.665,A -85,B 0,C 180,E1 -9991.081,E2 -9991.081} C_VEL
LIN {X 0,Y 423.589,Z 352.671,A -85,B 0,C 180,E1 -9991.865,E2 -9991.865} C_VEL
LIN {X 0,Y 420.687,Z 353.75,A -85,B 0,C 180,E1 -9993.145,E2 -9993.145} C_VEL
LIN {X 0,Y 418.266,Z 354.152,A -85,B 0,C 180,E1 -9994.183,E2 -9994.183} C_VEL
LIN {X 0,Y 417.21,Z 354.028,A -85,B 0,C 180,E1 -9995.121,E2 -9995.121} C_VEL
LIN {X 0,Y 417.199,Z 353.929,A -85,B 0,C 180,E1 -9995.257,E2 -9995.257} C_VEL
LIN {X 0,Y 417.308,Z 352.816,A -85,B 0,C 180,E1 -9996.769,E2 -9996.769} C_VEL
LIN {X 0,Y 417.455,Z 349.909,A -85,B 0,C 180,E1 -9998.713,E2 -9998.713} C_VEL
LIN {X 0,Y 417.654,Z 346.57,A -85,B 0,C 180,E1 -10000.175,E2 -10000.175} C_VEL
LIN {X 0,Y 418.018,Z 342.147,A -85,B 0,C 180,E1 -10001.638,E2 -10001.638} C_VEL
LIN {X 0,Y 418.511,Z 336.046,A -85,B 0,C 180,E1 -10003.208,E2 -10003.208} C_VEL
LIN {X 0,Y 419.057,Z 329.408,A -85,B 0,C 180,E1 -10004.569,E2 -10004.569} C_VEL
LIN {X 0,Y 419.833,Z 320.536,A -85,B 0,C 180,E1 -10006.033,E2 -10006.033} C_VEL
LIN {X 0,Y 420.582,Z 311.401,A -85,B 0,C 180,E1 -10007.252,E2 -10007.252} C_VEL
LIN {X 0,Y 421.248,Z 301.11,A -85,B 0,C 180,E1 -10008.363,E2 -10008.363} C_VEL
LIN {X 0,Y 422.044,Z 289.843,A -85,B 0,C 180,E1 -10009.326,E2 -10009.326} C_VEL
LIN {X 0,Y 422.614,Z 277.317,A -85,B 0,C 180,E1 -10010.162,E2 -10010.162} C_VEL
LIN {X 0,Y 422.819,Z 272.361,A -85,B 0,C 180,E1 -10010.428,E2 -10010.428} C_VEL
LIN {X 0,Y 420.112,Z 260.858,A -85,B 0,C 180,E1 -10011.065,E2 -10011.065} C_VEL
LIN {X 0,Y 417.425,Z 251.334,A -85,B 0,C 180,E1 -10011.52,E2 -10011.52} C_VEL
LIN {X 0,Y 417.545,Z 247.795,A -85,B 0,C 180,E1 -10014.883,E2 -10014.883} C_VEL
LIN {X 0,Y 417.632,Z 244.531,A -85,B 0,C 180,E1 -10018.11,E2 -10018.11} C_VEL
LIN {X 0,Y 417.671,Z 241.294,A -85,B 0,C 180,E1 -10021.439,E2 -10021.439} C_VEL
LIN {X 0,Y 417.811,Z 238.012,A -85,B 0,C 180,E1 -10024.882,E2 -10024.882} C_VEL
LIN {X 0,Y 417.856,Z 236.823,A -85,B 0,C 180,E1 -10026.164,E2 -10026.164} C_VEL
LIN {X 0,Y 418.025,Z 236.416,A -85,B 0,C 180,E1 -10027.797,E2 -10027.797} C_VEL
LIN {X 0,Y 418.203,Z 236.393,A -85,B 0,C 180,E1 -10030.948,E2 -10030.948} C_VEL
LIN {X 0,Y 418.203,Z 236.392,A -85,B 0,C 180,E1 -10033.728,E2 -10033.728} C_VEL
LIN {X 0,Y 418.2,Z 236.393,A -85,B 0,C 180,E1 -10036.447,E2 -10036.447} C_VEL
LIN {X 0,Y 418.213,Z 236.392,A -85,B 0,C 180,E1 -10039.129,E2 -10039.129} C_VEL
LIN {X 0,Y 418.224,Z 236.389,A -85,B 0,C 180,E1 -10042.165,E2 -10042.165} C_VEL
LIN {X 0,Y 418.257,Z 236.385,A -85,B 0,C 180,E1 -10045.418,E2 -10045.418} C_VEL
LIN {X 0,Y 418.201,Z 236.391,A -85,B 0,C 180,E1 -10048.603,E2 -10048.603} C_VEL
LIN {X 0,Y 418.282,Z 236.381,A -85,B 0,C 180,E1 -10051.936,E2 -10051.936} C_VEL
LIN {X 0,Y 418.28,Z 236.381,A -85,B 0,C 180,E1 -10055.162,E2 -10055.162} C_VEL
LIN {X 0,Y 418.223,Z 236.388,A -85,B 0,C 180,E1 -10058.303,E2 -10058.303} C_VEL
LIN {X 0,Y 418.272,Z 236.381,A -85,B 0,C 180,E1 -10061.382,E2 -10061.382} C_VEL
LIN {X 0,Y 418.291,Z 236.381,A -85,B 0,C 180,E1 -10064.405,E2 -10064.405} C_VEL
LIN {X 0,Y 418.344,Z 236.377,A -85,B 0,C 180,E1 -10067.385,E2 -10067.385} C_VEL
LIN {X 0,Y 418.388,Z 236.367,A -85,B 0,C 180,E1 -10071.305,E2 -10071.305} C_VEL
LIN {X 0,Y 418.524,Z 236.353,A -85,B 0,C 180,E1 -10074.217,E2 -10074.217} C_VEL
LIN {X 0,Y 418.534,Z 236.349,A -85,B 0,C 180,E1 -10078.075,E2 -10078.075} C_VEL
LIN {X 0,Y 418.657,Z 236.335,A -85,B 0,C 180,E1 -10080,E2 -10080} C_VEL
LIN {X 0,Y 418.5,Z 236.354,A -85,B 0,C 180,E1 -10082.888,E2 -10082.888} C_VEL
LIN {X 0,Y 418.523,Z 236.352,A -85,B 0,C 180,E1 -10085.783,E2 -10085.783} C_VEL
LIN {X 0,Y 418.388,Z 236.371,A -85,B 0,C 180,E1 -10088.695,E2 -10088.695} C_VEL
LIN {X 0,Y 418.303,Z 236.379,A -85,B 0,C 180,E1 -10091.631,E2 -10091.631} C_VEL
LIN {X 0,Y 418.291,Z 236.379,A -85,B 0,C 180,E1 -10094.597,E2 -10094.597} C_VEL
LIN {X 0,Y 418.277,Z 236.381,A -85,B 0,C 180,E1 -10097.604,E2 -10097.604} C_VEL
LIN {X 0,Y 418.238,Z 236.388,A -85,B 0,C 180,E1 -10100.664,E2 -10100.664} C_VEL
LIN {X 0,Y 418.276,Z 236.384,A -85,B 0,C 180,E1 -10103.782,E2 -10103.782} C_VEL
LIN {X 0,Y 418.299,Z 236.381,A -85,B 0,C 180,E1 -10107.071,E2 -10107.071} C_VEL
LIN {X 0,Y 418.252,Z 236.389,A -85,B 0,C 180,E1 -10110.272,E2 -10110.272} C_VEL
LIN {X 0,Y 418.239,Z 236.39,A -85,B 0,C 180,E1 -10113.678,E2 -10113.678} C_VEL
LIN {X 0,Y 418.231,Z 236.387,A -85,B 0,C 180,E1 -10117.225,E2 -10117.225} C_VEL
LIN {X 0,Y 418.239,Z 236.387,A -85,B 0,C 180,E1 -10119.683,E2 -10119.683} C_VEL
LIN {X 0,Y 418.215,Z 236.39,A -85,B 0,C 180,E1 -10122.321,E2 -10122.321} C_VEL
LIN {X 0,Y 418.228,Z 236.391,A -85,B 0,C 180,E1 -10125.11,E2 -10125.11} C_VEL
LIN {X 0,Y 418.26,Z 236.559,A -85,B 0,C 180,E1 -10126.689,E2 -10126.689} C_VEL
LIN {X 0,Y 419.352,Z 242.292,A -85,B 0,C 180,E1 -10129.82,E2 -10129.82} C_VEL
LIN {X 0,Y 420.398,Z 248.606,A -85,B 0,C 180,E1 -10133.001,E2 -10133.001} C_VEL
LIN {X 0,Y 420.401,Z 252.897,A -85,B 0,C 180,E1 -10135,E2 -10135} C_VEL
LIN {X 0,Y 419.821,Z 260.142,A -85,B 0,C 180,E1 -10138.178,E2 -10138.178} C_VEL
LIN {X 0,Y 419.202,Z 269.244,A -85,B 0,C 180,E1 -10142.005,E2 -10142.005} C_VEL
LIN {X 0,Y 418.642,Z 277.09,A -85,B 0,C 180,E1 -10145.187,E2 -10145.187} C_VEL
LIN {X 0,Y 418.271,Z 284.934,A -85,B 0,C 180,E1 -10148.307,E2 -10148.307} C_VEL
LIN {X 0,Y 417.909,Z 292.789,A -85,B 0,C 180,E1 -10151.367,E2 -10151.367} C_VEL
LIN {X 0,Y 417.737,Z 296.202,A -85,B 0,C 180,E1 -10152.686,E2 -10152.686} C_VEL
LIN {X 0,Y 420.113,Z 311.226,A -85,B 0,C 180,E1 -10153.254,E2 -10153.254} C_VEL
LIN {X 0,Y 421.78,Z 322.866,A -85,B 0,C 180,E1 -10153.857,E2 -10153.857} C_VEL
LIN {X 0,Y 421.211,Z 333.949,A -85,B 0,C 180,E1 -10154.518,E2 -10154.518} C_VEL
LIN {X 0,Y 420.401,Z 346.418,A -85,B 0,C 180,E1 -10155.479,E2 -10155.479} C_VEL
LIN {X 0,Y 419.671,Z 357.364,A -85,B 0,C 180,E1 -10156.566,E2 -10156.566} C_VEL
LIN {X 0,Y 419.124,Z 366.304,A -85,B 0,C 180,E1 -10157.657,E2 -10157.657} C_VEL
LIN {X 0,Y 418.381,Z 376.022,A -85,B 0,C 180,E1 -10159.108,E2 -10159.108} C_VEL
LIN {X 0,Y 417.858,Z 383.769,A -85,B 0,C 180,E1 -10160.563,E2 -10160.563} C_VEL
LIN {X 0,Y 417.538,Z 389.082,A -85,B 0,C 180,E1 -10161.776,E2 -10161.776} C_VEL
LIN {X 0,Y 417.277,Z 395.251,A -85,B 0,C 180,E1 -10163.571,E2 -10163.571} C_VEL
LIN {X 0,Y 417.161,Z 399.326,A -85,B 0,C 180,E1 -10165.169,E2 -10165.169} C_VEL
LIN {X 0,Y 417.035,Z 401.201,A -85,B 0,C 180,E1 -10166.136,E2 -10166.136} C_VEL
LIN {X 0,Y 417.106,Z 402.618,A -85,B 0,C 180,E1 -10167.104,E2 -10167.104} C_VEL
LIN {X 0,Y 417.035,Z 404.238,A -85,B 0,C 180,E1 -10169.036,E2 -10169.036} C_VEL
LIN {X 0,Y 417.047,Z 404.459,A -85,B 0,C 180,E1 -10170.001,E2 -10170.001} C_VEL
LIN {X 0,Y 417.035,Z 404.241,A -85,B 0,C 180,E1 -10170.967,E2 -10170.967} C_VEL
LIN {X 0,Y 417.107,Z 402.628,A -85,B 0,C 180,E1 -10172.899,E2 -10172.899} C_VEL
LIN {X 0,Y 417.035,Z 401.213,A -85,B 0,C 180,E1 -10173.867,E2 -10173.867} C_VEL
LIN {X 0,Y 417.193,Z 398.257,A -85,B 0,C 180,E1 -10175.318,E2 -10175.318} C_VEL
LIN {X 0,Y 417.277,Z 394.247,A -85,B 0,C 180,E1 -10176.772,E2 -10176.772} C_VEL
LIN {X 0,Y 417.59,Z 388.092,A -85,B 0,C 180,E1 -10178.47,E2 -10178.47} C_VEL
LIN {X 0,Y 418.017,Z 381.373,A -85,B 0,C 180,E1 -10179.925,E2 -10179.925} C_VEL
LIN {X 0,Y 418.596,Z 373.044,A -85,B 0,C 180,E1 -10181.379,E2 -10181.379} C_VEL
LIN {X 0,Y 419.215,Z 364.512,A -85,B 0,C 180,E1 -10182.589,E2 -10182.589} C_VEL
LIN {X 0,Y 419.958,Z 353.583,A -85,B 0,C 180,E1 -10183.839,E2 -10183.839} C_VEL
LIN {X 0,Y 420.685,Z 342.119,A -85,B 0,C 180,E1 -10184.885,E2 -10184.885} C_VEL
LIN {X 0,Y 421.455,Z 330.207,A -85,B 0,C 180,E1 -10185.724,E2 -10185.724} C_VEL
LIN {X 0,Y 421.744,Z 322.771,A -85,B 0,C 180,E1 -10186.147,E2 -10186.147} C_VEL
LIN {X 0,Y 419.896,Z 309.607,A -85,B 0,C 180,E1 -10186.808,E2 -10186.808} C_VEL
LIN {X 0,Y 417.732,Z 296.267,A -85,B 0,C 180,E1 -10187.288,E2 -10187.288} C_VEL
LIN {X 0,Y 418.065,Z 288.825,A -85,B 0,C 180,E1 -10190.16,E2 -10190.16} C_VEL
LIN {X 0,Y 418.427,Z 280.866,A -85,B 0,C 180,E1 -10193.249,E2 -10193.249} C_VEL
LIN {X 0,Y 418.919,Z 272.894,A -85,B 0,C 180,E1 -10196.398,E2 -10196.398} C_VEL
LIN {X 0,Y 419.314,Z 265.538,A -85,B 0,C 180,E1 -10199.36,E2 -10199.36} C_VEL
LIN {X 0,Y 419.84,Z 258.226,A -85,B 0,C 180,E1 -10202.391,E2 -10202.391} C_VEL
LIN {X 0,Y 420.307,Z 252.205,A -85,B 0,C 180,E1 -10204.982,E2 -10204.982} C_VEL
LIN {X 0,Y 420.235,Z 247.681,A -85,B 0,C 180,E1 -10207.019,E2 -10207.019} C_VEL
LIN {X 0,Y 419.121,Z 241.1,A -85,B 0,C 180,E1 -10210.21,E2 -10210.21} C_VEL
LIN {X 0,Y 418.29,Z 236.385,A -85,B 0,C 180,E1 -10212.733,E2 -10212.733} C_VEL
LIN {X 0,Y 418.217,Z 236.394,A -85,B 0,C 180,E1 -10216.271,E2 -10216.271} C_VEL
LIN {X 0,Y 418.23,Z 236.391,A -85,B 0,C 180,E1 -10219.131,E2 -10219.131} C_VEL
LIN {X 0,Y 418.232,Z 236.388,A -85,B 0,C 180,E1 -10222.168,E2 -10222.168} C_VEL
LIN {X 0,Y 418.259,Z 236.381,A -85,B 0,C 180,E1 -10225.423,E2 -10225.423} C_VEL
LIN {X 0,Y 418.216,Z 236.391,A -85,B 0,C 180,E1 -10228.604,E2 -10228.604} C_VEL
LIN {X 0,Y 418.268,Z 236.384,A -85,B 0,C 180,E1 -10231.935,E2 -10231.935} C_VEL
LIN {X 0,Y 418.279,Z 236.381,A -85,B 0,C 180,E1 -10235.162,E2 -10235.162} C_VEL
LIN {X 0,Y 418.242,Z 236.389,A -85,B 0,C 180,E1 -10238.304,E2 -10238.304} C_VEL
LIN {X 0,Y 418.277,Z 236.381,A -85,B 0,C 180,E1 -10241.383,E2 -10241.383} C_VEL
LIN {X 0,Y 418.257,Z 236.385,A -85,B 0,C 180,E1 -10244.404,E2 -10244.404} C_VEL
LIN {X 0,Y 418.36,Z 236.371,A -85,B 0,C 180,E1 -10247.386,E2 -10247.386} C_VEL
LIN {X 0,Y 418.381,Z 236.37,A -85,B 0,C 180,E1 -10251.305,E2 -10251.305} C_VEL
LIN {X 0,Y 418.512,Z 236.354,A -85,B 0,C 180,E1 -10254.217,E2 -10254.217} C_VEL
LIN {X 0,Y 418.549,Z 236.349,A -85,B 0,C 180,E1 -10258.076,E2 -10258.076} C_VEL
LIN {X 0,Y 418.674,Z 236.334,A -85,B 0,C 180,E1 -10260,E2 -10260} C_VEL
LIN {X 0,Y 418.495,Z 236.355,A -85,B 0,C 180,E1 -10262.888,E2 -10262.888} C_VEL
LIN {X 0,Y 418.442,Z 236.36,A -85,B 0,C 180,E1 -10266.752,E2 -10266.752} C_VEL
LIN {X 0,Y 418.338,Z 236.374,A -85,B 0,C 180,E1 -10269.672,E2 -10269.672} C_VEL
LIN {X 0,Y 418.355,Z 236.375,A -85,B 0,C 180,E1 -10273,E2 -10273} C_VEL
LIN {X 0,Y 418.321,Z 236.379,A -85,B 0,C 180,E1 -10276.735,E2 -10276.735} C_VEL
LIN {X 0,Y 418.278,Z 236.381,A -85,B 0,C 180,E1 -10279.79,E2 -10279.79} C_VEL
LIN {X 0,Y 418.234,Z 236.389,A -85,B 0,C 180,E1 -10282.737,E2 -10282.737} C_VEL
LIN {X 0,Y 418.217,Z 236.387,A -85,B 0,C 180,E1 -10285.908,E2 -10285.908} C_VEL
LIN {X 0,Y 418.264,Z 236.383,A -85,B 0,C 180,E1 -10289.162,E2 -10289.162} C_VEL
LIN {X 0,Y 418.265,Z 236.385,A -85,B 0,C 180,E1 -10292.843,E2 -10292.843} C_VEL
LIN {X 0,Y 418.251,Z 236.388,A -85,B 0,C 180,E1 -10296.237,E2 -10296.237} C_VEL
LIN {X 0,Y 418.249,Z 236.385,A -85,B 0,C 180,E1 -10299.683,E2 -10299.683} C_VEL
LIN {X 0,Y 418.231,Z 236.39,A -85,B 0,C 180,E1 -10302.32,E2 -10302.32} C_VEL
LIN {X 0,Y 418.241,Z 236.384,A -85,B 0,C 180,E1 -10305.108,E2 -10305.108} C_VEL
LIN {X 0,Y 418.224,Z 236.389,A -85,B 0,C 180,E1 -10307.763,E2 -10307.763} C_VEL
LIN {X 0,Y 418.243,Z 236.387,A -85,B 0,C 180,E1 -10311.556,E2 -10311.556} C_VEL
LIN {X 0,Y 418.257,Z 236.384,A -85,B 0,C 180,E1 -10315.157,E2 -10315.157} C_VEL
LIN {X 0,Y 418.208,Z 236.393,A -85,B 0,C 180,E1 -10317.467,E2 -10317.467} C_VEL
LIN {X 0,Y 417.924,Z 236.426,A -85,B 0,C 180,E1 -10320.811,E2 -10320.811} C_VEL
LIN {X 0,Y 417.681,Z 236.797,A -85,B 0,C 180,E1 -10322.978,E2 -10322.978} C_VEL
LIN {X 0,Y 417.595,Z 239.895,A -85,B 0,C 180,E1 -10326.176,E2 -10326.176} C_VEL
LIN {X 0,Y 417.513,Z 243.012,A -85,B 0,C 180,E1 -10329.298,E2 -10329.298} C_VEL
LIN {X 0,Y 417.479,Z 246.166,A -85,B 0,C 180,E1 -10332.36,E2 -10332.36} C_VEL
LIN {X 0,Y 417.441,Z 249.37,A -85,B 0,C 180,E1 -10335.371,E2 -10335.371} C_VEL
LIN {X 0,Y 417.497,Z 251.333,A -85,B 0,C 180,E1 -10337.03,E2 -10337.03} C_VEL
LIN {X 0,Y 420.714,Z 264.523,A -85,B 0,C 180,E1 -10337.598,E2 -10337.598} C_VEL
LIN {X 0,Y 422.169,Z 272.2,A -85,B 0,C 180,E1 -10338.006,E2 -10338.006} C_VEL
LIN {X 0,Y 421.681,Z 284.151,A -85,B 0,C 180,E1 -10338.705,E2 -10338.705} C_VEL
LIN {X 0,Y 421.049,Z 295.195,A -85,B 0,C 180,E1 -10339.54,E2 -10339.54} C_VEL
LIN {X 0,Y 420.482,Z 304.833,A -85,B 0,C 180,E1 -10340.45,E2 -10340.45} C_VEL
LIN {X 0,Y 419.936,Z 314.56,A -85,B 0,C 180,E1 -10341.578,E2 -10341.578} C_VEL
LIN {X 0,Y 419.275,Z 323.039,A -85,B 0,C 180,E1 -10342.776,E2 -10342.776} C_VEL
LIN {X 0,Y 418.603,Z 331.274,A -85,B 0,C 180,E1 -10344.217,E2 -10344.217} C_VEL
LIN {X 0,Y 418.11,Z 337.907,A -85,B 0,C 180,E1 -10345.661,E2 -10345.661} C_VEL
LIN {X 0,Y 417.622,Z 343.216,A -85,B 0,C 180,E1 -10347.105,E2 -10347.105} C_VEL
LIN {X 0,Y 417.395,Z 347.355,A -85,B 0,C 180,E1 -10348.551,E2 -10348.551} C_VEL
LIN {X 0,Y 417.222,Z 350.458,A -85,B 0,C 180,E1 -10349.999,E2 -10349.999} C_VEL
LIN {X 0,Y 417.215,Z 352.117,A -85,B 0,C 180,E1 -10351.064,E2 -10351.064} C_VEL
LIN {X 0,Y 417.219,Z 353.127,A -85,B 0,C 180,E1 -10351.929,E2 -10351.929} C_VEL
LIN {X 0,Y 417.264,Z 353.831,A -85,B 0,C 180,E1 -10352.895,E2 -10352.895} C_VEL
LIN {X 0,Y 417.176,Z 354.124,A -85,B 0,C 180,E1 -10354.83,E2 -10354.83} C_VEL
LIN {X 0,Y 417.199,Z 353.929,A -85,B 0,C 180,E1 -10355.257,E2 -10355.257} C_VEL
LIN {X 0,Y 416.591,Z 353.528,A -85,B 0,C 180,E1 -10356.062,E2 -10356.062} C_VEL
LIN {X 0,Y 413.802,Z 352.386,A -85,B 0,C 180,E1 -10357.368,E2 -10357.368} C_VEL
LIN {X 0,Y 411.466,Z 350.994,A -85,B 0,C 180,E1 -10358.41,E2 -10358.41} C_VEL
LIN {X 0,Y 410.525,Z 349.555,A -85,B 0,C 180,E1 -10359.202,E2 -10359.202} C_VEL
LIN {X 0,Y 410.485,Z 348.979,A -85,B 0,C 180,E1 -10359.466,E2 -10359.466} C_VEL
LIN {X 0,Y 410.715,Z 345.499,A -85,B 0,C 180,E1 -10360.848,E2 -10360.848} C_VEL
LIN {X 0,Y 411.168,Z 340.645,A -85,B 0,C 180,E1 -10362.335,E2 -10362.335} C_VEL
LIN {X 0,Y 411.707,Z 334.512,A -85,B 0,C 180,E1 -10363.825,E2 -10363.825} C_VEL
LIN {X 0,Y 412.367,Z 326.84,A -85,B 0,C 180,E1 -10365.316,E2 -10365.316} C_VEL
LIN {X 0,Y 413.071,Z 318.954,A -85,B 0,C 180,E1 -10366.556,E2 -10366.556} C_VEL
LIN {X 0,Y 413.888,Z 309.301,A -85,B 0,C 180,E1 -10367.795,E2 -10367.795} C_VEL
LIN {X 0,Y 414.674,Z 298.54,A -85,B 0,C 180,E1 -10368.912,E2 -10368.912} C_VEL
LIN {X 0,Y 415.426,Z 288.043,A -85,B 0,C 180,E1 -10369.775,E2 -10369.775} C_VEL
LIN {X 0,Y 415.942,Z 275.574,A -85,B 0,C 180,E1 -10370.574,E2 -10370.574} C_VEL
LIN {X 0,Y 415.999,Z 273.174,A -85,B 0,C 180,E1 -10370.707,E2 -10370.707} C_VEL
LIN {X 0,Y 413.05,Z 261.136,A -85,B 0,C 180,E1 -10371.396,E2 -10371.396} C_VEL
LIN {X 0,Y 410.401,Z 251.777,A -85,B 0,C 180,E1 -10371.833,E2 -10371.833} C_VEL
LIN {X 0,Y 410.498,Z 248.131,A -85,B 0,C 180,E1 -10375.34,E2 -10375.34} C_VEL
LIN {X 0,Y 410.589,Z 244.839,A -85,B 0,C 180,E1 -10378.636,E2 -10378.636} C_VEL
LIN {X 0,Y 410.646,Z 241.576,A -85,B 0,C 180,E1 -10382.041,E2 -10382.041} C_VEL
LIN {X 0,Y 410.781,Z 238.262,A -85,B 0,C 180,E1 -10385.568,E2 -10385.568} C_VEL
LIN {X 0,Y 410.84,Z 237.313,A -85,B 0,C 180,E1 -10386.776,E2 -10386.776} C_VEL
LIN {X 0,Y 411.116,Z 237.275,A -85,B 0,C 180,E1 -10389.711,E2 -10389.711} C_VEL
LIN {X 0,Y 411.166,Z 237.269,A -85,B 0,C 180,E1 -10393.132,E2 -10393.132} C_VEL
LIN {X 0,Y 411.16,Z 237.271,A -85,B 0,C 180,E1 -10395.88,E2 -10395.88} C_VEL
LIN {X 0,Y 411.152,Z 237.27,A -85,B 0,C 180,E1 -10398.771,E2 -10398.771} C_VEL
LIN {X 0,Y 411.189,Z 237.265,A -85,B 0,C 180,E1 -10402.025,E2 -10402.025} C_VEL
LIN {X 0,Y 411.198,Z 237.266,A -85,B 0,C 180,E1 -10405.665,E2 -10405.665} C_VEL
LIN {X 0,Y 411.18,Z 237.266,A -85,B 0,C 180,E1 -10409.151,E2 -10409.151} C_VEL
LIN {X 0,Y 411.249,Z 237.257,A -85,B 0,C 180,E1 -10412.521,E2 -10412.521} C_VEL
LIN {X 0,Y 411.217,Z 237.264,A -85,B 0,C 180,E1 -10415.784,E2 -10415.784} C_VEL
LIN {X 0,Y 411.186,Z 237.269,A -85,B 0,C 180,E1 -10418.965,E2 -10418.965} C_VEL
LIN {X 0,Y 411.241,Z 237.259,A -85,B 0,C 180,E1 -10422.084,E2 -10422.084} C_VEL
LIN {X 0,Y 411.249,Z 237.258,A -85,B 0,C 180,E1 -10425.147,E2 -10425.147} C_VEL
LIN {X 0,Y 411.271,Z 237.254,A -85,B 0,C 180,E1 -10428.167,E2 -10428.167} C_VEL
LIN {X 0,Y 411.47,Z 237.233,A -85,B 0,C 180,E1 -10432.146,E2 -10432.146} C_VEL
LIN {X 0,Y 411.483,Z 237.231,A -85,B 0,C 180,E1 -10434.118,E2 -10434.118} C_VEL
LIN {X 0,Y 411.503,Z 237.225,A -85,B 0,C 180,E1 -10438.042,E2 -10438.042} C_VEL
LIN {X 0,Y 411.626,Z 237.211,A -85,B 0,C 180,E1 -10440,E2 -10440} C_VEL
LIN {X 0,Y 411.456,Z 237.231,A -85,B 0,C 180,E1 -10442.937,E2 -10442.937} C_VEL
LIN {X 0,Y 411.482,Z 237.229,A -85,B 0,C 180,E1 -10445.882,E2 -10445.882} C_VEL
LIN {X 0,Y 411.47,Z 237.23,A -85,B 0,C 180,E1 -10447.853,E2 -10447.853} C_VEL
LIN {X 0,Y 411.271,Z 237.256,A -85,B 0,C 180,E1 -10451.833,E2 -10451.833} C_VEL
LIN {X 0,Y 411.248,Z 237.257,A -85,B 0,C 180,E1 -10454.853,E2 -10454.853} C_VEL
LIN {X 0,Y 411.241,Z 237.258,A -85,B 0,C 180,E1 -10457.916,E2 -10457.916} C_VEL
LIN {X 0,Y 411.185,Z 237.265,A -85,B 0,C 180,E1 -10461.035,E2 -10461.035} C_VEL
LIN {X 0,Y 411.216,Z 237.261,A -85,B 0,C 180,E1 -10464.216,E2 -10464.216} C_VEL
LIN {X 0,Y 411.249,Z 237.257,A -85,B 0,C 180,E1 -10467.478,E2 -10467.478} C_VEL
LIN {X 0,Y 411.189,Z 237.265,A -85,B 0,C 180,E1 -10470.848,E2 -10470.848} C_VEL
LIN {X 0,Y 411.196,Z 237.265,A -85,B 0,C 180,E1 -10474.335,E2 -10474.335} C_VEL
LIN {X 0,Y 411.185,Z 237.265,A -85,B 0,C 180,E1 -10477.975,E2 -10477.975} C_VEL
LIN {X 0,Y 411.17,Z 237.268,A -85,B 0,C 180,E1 -10480.506,E2 -10480.506} C_VEL
LIN {X 0,Y 411.163,Z 237.271,A -85,B 0,C 180,E1 -10483.135,E2 -10483.135} C_VEL
LIN {X 0,Y 411.187,Z 237.426,A -85,B 0,C 180,E1 -10486.272,E2 -10486.272} C_VEL
LIN {X 0,Y 412.366,Z 243.448,A -85,B 0,C 180,E1 -10489.638,E2 -10489.638} C_VEL
LIN {X 0,Y 413.457,Z 250.031,A -85,B 0,C 180,E1 -10493.027,E2 -10493.027} C_VEL
LIN {X 0,Y 413.373,Z 254.816,A -85,B 0,C 180,E1 -10495.283,E2 -10495.283} C_VEL
LIN {X 0,Y 412.768,Z 261.723,A -85,B 0,C 180,E1 -10498.356,E2 -10498.356} C_VEL
